C05493=1186.464,-67.586,-41.401,179.419,5.670,149.176
C05494=1186.458,-67.337,-41.411,179.422,5.670,149.175
C05495=1186.453,-67.087,-41.423,179.424,5.671,149.175
C05496=1186.448,-66.837,-41.433,179.426,5.671,149.174
C05497=1186.442,-66.588,-41.445,179.429,5.671,149.173
C05498=1186.438,-66.338,-41.456,179.431,5.672,149.173
C05499=1186.432,-66.088,-41.466,179.433,5.672,149.172
C05500=1186.427,-65.839,-41.477,179.436,5.672,149.171
C05501=1186.422,-65.589,-41.489,179.438,5.673,149.171
C05502=1186.416,-65.339,-41.500,179.440,5.672,149.170
C05503=1186.412,-65.090,-41.511,179.443,5.673,149.169
C05504=1186.406,-64.839,-41.522,179.445,5.674,149.169
C05505=1186.401,-64.590,-41.533,179.447,5.673,149.168
C05506=1186.396,-64.341,-41.544,179.450,5.674,149.168
C05507=1186.391,-64.090,-41.555,179.452,5.675,149.167
C05508=1186.385,-63.841,-41.566,179.454,5.674,149.166
C05509=1186.380,-63.591,-41.578,179.457,5.675,149.166
C05510=1186.376,-63.342,-41.589,179.459,5.675,149.165
C05511=1186.369,-63.092,-41.600,179.461,5.675,149.164
C05512=1186.365,-62.842,-41.611,179.464,5.675,149.164
C05513=1186.360,-62.593,-41.622,179.466,5.676,149.163
C05514=1186.354,-62.342,-41.633,179.468,5.676,149.163
C05515=1186.349,-62.093,-41.644,179.471,5.676,149.162
C05516=1186.344,-61.844,-41.656,179.473,5.677,149.161
C05517=1186.339,-61.594,-41.668,179.475,5.677,149.161
C05518=1186.333,-61.344,-41.678,179.478,5.677,149.160
C05519=1186.328,-61.094,-41.690,179.480,5.678,149.159
C05520=1186.323,-60.845,-41.701,179.482,5.677,149.159
C05521=1186.318,-60.595,-41.712,179.485,5.678,149.158
C05522=1186.312,-60.345,-41.723,179.487,5.678,149.157
C05523=1186.307,-60.095,-41.734,179.489,5.678,149.157
C05524=1186.302,-59.846,-41.746,179.491,5.679,149.156
C05525=1186.297,-59.596,-41.757,179.494,5.679,149.156
C05526=1186.292,-59.347,-41.768,179.497,5.680,149.155
C05527=1186.286,-59.096,-41.780,179.498,5.680,149.154
C05528=1186.281,-58.847,-41.791,179.501,5.680,149.154
C05529=1186.275,-58.598,-41.802,179.504,5.681,149.153
C05530=1186.271,-58.348,-41.814,179.506,5.680,149.152
C05531=1186.266,-58.098,-41.825,179.508,5.681,149.152
C05532=1186.261,-57.848,-41.837,179.511,5.681,149.151
C05533=1186.256,-57.598,-41.847,179.513,5.681,149.150
C05534=1186.250,-57.349,-41.859,179.515,5.682,149.150
C05535=1186.245,-57.099,-41.870,179.518,5.682,149.149
C05536=1186.239,-56.849,-41.882,179.520,5.683,149.148
C05537=1186.235,-56.600,-41.893,179.522,5.683,149.148
C05538=1186.229,-56.351,-41.905,179.525,5.683,149.147
C05539=1186.224,-56.101,-41.916,179.527,5.684,149.147
C05540=1186.219,-55.851,-41.928,179.529,5.683,149.146
C05541=1186.214,-55.601,-41.939,179.531,5.684,149.145
C05542=1186.209,-55.352,-41.951,179.534,5.685,149.145
C05543=1186.203,-55.102,-41.961,179.536,5.684,149.144
C05544=1186.198,-54.852,-41.973,179.538,5.685,149.144
C05545=1186.193,-54.602,-41.985,179.541,5.685,149.143
C05546=1186.188,-54.353,-41.996,179.544,5.686,149.142
C05547=1186.183,-54.103,-42.008,179.546,5.685,149.141
C05548=1186.178,-53.853,-42.019,179.548,5.686,149.141
C05549=1186.172,-53.604,-42.031,179.551,5.687,149.140
C05550=1186.166,-53.354,-42.043,179.553,5.686,149.140
C05551=1186.162,-53.104,-42.054,179.555,5.687,149.139
C05552=1186.156,-52.854,-42.066,179.558,5.688,149.138
C05553=1186.152,-52.605,-42.077,179.560,5.688,149.138
C05554=1186.146,-52.355,-42.089,179.562,5.688,149.137
C05555=1186.141,-52.106,-42.100,179.564,5.688,149.136
C05556=1186.136,-51.856,-42.112,179.567,5.689,149.136
C05557=1186.131,-51.606,-42.123,179.569,5.689,149.135
C05558=1186.125,-51.356,-42.135,179.571,5.689,149.135
C05559=1186.120,-51.106,-42.147,179.574,5.690,149.134
C05560=1186.115,-50.857,-42.158,179.577,5.690,149.133
C05561=1186.110,-50.607,-42.171,179.579,5.690,149.132
C05562=1186.105,-50.359,-42.182,179.581,5.691,149.132
C05563=1186.099,-50.109,-42.193,179.584,5.691,149.131
C05564=1186.094,-49.838,-42.206,179.586,5.692,149.131
C05565=1186.088,-49.568,-42.218,179.589,5.692,149.130
C05566=1186.083,-49.298,-42.231,179.591,5.692,149.129
C05567=1186.077,-49.027,-42.244,179.594,5.692,149.128
C05568=1186.072,-48.777,-42.256,179.596,5.693,149.128
C05569=1186.067,-48.528,-42.267,179.599,5.693,149.127
C05570=1186.061,-48.278,-42.279,179.601,5.693,149.127
C05571=1186.056,-48.029,-42.291,179.603,5.693,149.126
C05572=1186.051,-47.779,-42.302,179.606,5.694,149.125
C05573=1186.046,-47.529,-42.314,179.608,5.695,149.125
C05574=1186.040,-47.280,-42.327,179.610,5.694,149.124
C05575=1186.036,-47.030,-42.338,179.613,5.695,149.123
C05576=1186.030,-46.780,-42.350,179.615,5.696,149.123
C05577=1186.025,-46.530,-42.362,179.618,5.696,149.122
C05578=1186.020,-46.281,-42.373,179.620,5.696,149.121
C05579=1186.015,-46.031,-42.386,179.622,5.696,149.121
C05580=1186.010,-45.781,-42.397,179.625,5.697,149.120
C05581=1186.004,-45.532,-42.408,179.627,5.697,149.120
C05582=1185.999,-45.282,-42.420,179.629,5.697,149.119
C05583=1185.994,-45.033,-42.432,179.632,5.698,149.118
C05584=1185.988,-44.783,-42.445,179.634,5.698,149.118
C05585=1185.984,-44.534,-42.456,179.637,5.699,149.117
C05586=1185.978,-44.284,-42.468,179.639,5.699,149.116
C05587=1185.973,-44.034,-42.480,179.641,5.699,149.116
C05588=1185.968,-43.784,-42.492,179.644,5.700,149.115
C05589=1185.963,-43.535,-42.504,179.647,5.700,149.114
C05590=1185.958,-43.285,-42.516,179.648,5.700,149.114
C05591=1185.952,-43.035,-42.528,179.651,5.700,149.113
C05592=1185.947,-42.786,-42.540,179.653,5.701,149.113
C05593=1185.942,-42.536,-42.551,179.656,5.701,149.112
C05594=1185.937,-42.286,-42.563,179.658,5.701,149.111
C05595=1185.932,-42.037,-42.576,179.660,5.702,149.111
C05596=1185.926,-41.787,-42.588,179.663,5.702,149.110
C05597=1185.922,-41.537,-42.599,179.665,5.703,149.109
C05598=1185.917,-41.288,-42.612,179.667,5.703,149.109
C05599=1185.911,-41.038,-42.623,179.670,5.703,149.108
C05600=1185.906,-40.788,-42.635,179.673,5.704,149.107
C05601=1185.901,-40.539,-42.648,179.675,5.704,149.107
C05602=1185.896,-40.289,-42.659,179.677,5.705,149.106
C05603=1185.891,-40.040,-42.672,179.680,5.704,149.105
C05604=1185.885,-39.790,-42.684,179.682,5.705,149.105
C05605=1185.880,-39.540,-42.696,179.684,5.706,149.104
C05606=1185.875,-39.290,-42.708,179.687,5.706,149.104
C05607=1185.869,-39.041,-42.720,179.689,5.706,149.103
C05608=1185.865,-38.792,-42.732,179.691,5.707,149.102
C05609=1185.860,-38.542,-42.744,179.694,5.707,149.102
C05610=1185.854,-38.292,-42.756,179.697,5.708,149.101
C05611=1185.849,-38.042,-42.768,179.699,5.708,149.100
C05612=1185.844,-37.792,-42.780,179.701,5.708,149.100
C05613=1185.838,-37.543,-42.793,179.704,5.708,149.099
C05614=1185.833,-37.293,-42.805,179.706,5.709,149.098
C05615=1185.828,-37.044,-42.817,179.709,5.709,149.098
C05616=1185.823,-36.794,-42.829,179.710,5.709,149.097
C05617=1185.818,-36.545,-42.841,179.713,5.710,149.097
C05618=1185.813,-36.294,-42.854,179.716,5.710,149.096
C05619=1185.808,-36.045,-42.866,179.718,5.711,149.095
C05620=1185.803,-35.795,-42.878,179.721,5.711,149.095
C05621=1185.798,-35.546,-42.891,179.723,5.711,149.094
C05622=1185.792,-35.296,-42.903,179.725,5.712,149.093
C05623=1185.787,-35.046,-42.915,179.728,5.712,149.093
C05624=1185.782,-34.796,-42.927,179.730,5.713,149.092
C05625=1185.776,-34.547,-42.940,179.733,5.713,149.091
C05626=1185.771,-34.297,-42.952,179.735,5.713,149.091
C05627=1185.766,-34.048,-42.964,179.737,5.714,149.090
C05628=1185.760,-33.798,-42.976,179.740,5.714,149.090
C05629=1185.755,-33.549,-42.989,179.742,5.715,149.089
C05630=1185.751,-33.299,-43.002,179.745,5.715,149.088
C05631=1185.745,-33.049,-43.013,179.747,5.715,149.088
C05632=1185.740,-32.799,-43.026,179.749,5.716,149.087
C05633=1185.735,-32.549,-43.038,179.752,5.716,149.086
C05634=1185.730,-32.300,-43.051,179.754,5.717,149.086
C05635=1185.725,-32.051,-43.063,179.757,5.717,149.085
C05636=1185.719,-31.801,-43.075,179.759,5.717,149.084
C05637=1185.714,-31.552,-43.088,179.762,5.717,149.084
C05638=1185.709,-31.302,-43.101,179.764,5.718,149.083
C05639=1185.704,-31.052,-43.112,179.766,5.719,149.083
C05640=1185.699,-30.802,-43.125,179.769,5.719,149.082
C05641=1185.694,-30.553,-43.138,179.771,5.719,149.081
C05642=1185.688,-30.303,-43.150,179.773,5.720,149.081
C05643=1185.683,-30.054,-43.162,179.776,5.720,149.080
C05644=1185.679,-29.804,-43.175,179.779,5.721,149.079
C05645=1185.673,-29.554,-43.187,179.781,5.721,149.079
C05646=1185.668,-29.304,-43.200,179.783,5.721,149.078
C05647=1185.663,-29.055,-43.212,179.786,5.721,149.077
C05648=1185.658,-28.805,-43.224,179.788,5.722,149.077
C05649=1185.653,-28.556,-43.237,179.790,5.723,149.076
C05650=1185.648,-28.306,-43.250,179.793,5.723,149.076
C05651=1185.643,-28.057,-43.262,179.796,5.724,149.075
C05652=1185.637,-27.807,-43.274,179.798,5.723,149.074
C05653=1185.632,-27.557,-43.287,179.800,5.724,149.074
C05654=1185.627,-27.308,-43.299,179.803,5.725,149.073
C05655=1185.622,-27.058,-43.313,179.805,5.725,149.072
C05656=1185.617,-26.808,-43.326,179.808,5.725,149.072
C05657=1185.611,-26.558,-43.337,179.810,5.726,149.071
C05658=1185.606,-26.309,-43.350,179.812,5.726,149.070
C05659=1185.601,-26.060,-43.363,179.815,5.726,149.070
C05660=1185.597,-25.810,-43.376,179.818,5.727,149.069
C05661=1185.591,-25.560,-43.388,179.820,5.728,149.069
C05662=1185.586,-25.310,-43.400,179.822,5.728,149.068
C05663=1185.581,-25.061,-43.413,179.825,5.729,149.067
C05664=1185.576,-24.811,-43.426,179.827,5.729,149.067
C05665=1185.571,-24.562,-43.439,179.829,5.729,149.066
C05666=1185.565,-24.312,-43.451,179.832,5.730,149.065
C05667=1185.560,-24.063,-43.464,179.835,5.730,149.065
C05668=1185.555,-23.793,-43.478,179.837,5.730,149.064
C05669=1185.550,-23.523,-43.492,179.840,5.731,149.063
C05670=1185.544,-23.253,-43.505,179.843,5.731,149.063
C05671=1185.538,-22.983,-43.519,179.845,5.732,149.062
C05672=1185.533,-22.734,-43.531,179.847,5.733,149.061
C05673=1185.528,-22.484,-43.544,179.850,5.733,149.061
C05674=1185.523,-22.235,-43.557,179.852,5.733,149.060
C05675=1185.517,-21.985,-43.570,179.854,5.734,149.060
C05676=1185.512,-21.736,-43.583,179.857,5.734,149.059
C05677=1185.508,-21.486,-43.596,179.860,5.735,149.058
C05678=1185.503,-21.236,-43.608,179.862,5.735,149.057
C05679=1185.497,-20.987,-43.622,179.865,5.736,149.057
C05680=1185.492,-20.737,-43.635,179.867,5.735,149.056
C05681=1185.487,-20.488,-43.647,179.869,5.736,149.056
C05682=1185.482,-20.238,-43.660,179.872,5.736,149.055
C05683=1185.476,-19.989,-43.673,179.874,5.737,149.054
C05684=1185.471,-19.739,-43.686,179.877,5.738,149.054
C05685=1185.466,-19.489,-43.699,179.879,5.738,149.053
C05686=1185.461,-19.240,-43.712,179.882,5.739,149.053
C05687=1185.456,-18.990,-43.725,179.884,5.739,149.052
C05688=1185.451,-18.740,-43.737,179.886,5.739,149.051
C05689=1185.446,-18.491,-43.750,179.889,5.740,149.051
C05690=1185.440,-18.241,-43.763,179.891,5.740,149.050
C05691=1185.435,-17.991,-43.776,179.894,5.741,149.049
C05692=1185.430,-17.742,-43.789,179.896,5.741,149.049
C05693=1185.425,-17.492,-43.802,179.899,5.742,149.048
C05694=1185.420,-17.242,-43.815,179.901,5.743,149.047
C05695=1185.415,-16.993,-43.827,179.903,5.742,149.047
C05696=1185.409,-16.743,-43.841,179.906,5.743,149.046
C05697=1185.405,-16.494,-43.854,179.909,5.743,149.045
C05698=1185.400,-16.245,-43.867,179.911,5.744,149.045
C05699=1185.394,-15.994,-43.880,179.914,5.744,149.044
C05700=1185.389,-15.745,-43.893,179.916,5.745,149.044
C05701=1185.385,-15.495,-43.906,179.918,5.746,149.043
C05702=1185.379,-15.245,-43.919,179.921,5.746,149.042
C05703=1185.374,-14.996,-43.932,179.924,5.747,149.042
C05704=1185.369,-14.746,-43.946,179.926,5.746,149.041
C05705=1185.364,-14.497,-43.959,179.928,5.747,149.041
C05706=1185.358,-14.248,-43.971,179.931,5.748,149.040
C05707=1185.353,-13.997,-43.985,179.933,5.748,149.039
C05708=1185.348,-13.748,-43.997,179.936,5.749,149.038
C05709=1185.344,-13.498,-44.010,179.938,5.749,149.038
C05710=1185.338,-13.249,-44.024,179.941,5.750,149.037
C05711=1185.333,-13.000,-44.037,179.943,5.750,149.037
C05712=1185.328,-12.749,-44.051,179.946,5.751,149.036
C05713=1185.322,-12.500,-44.063,179.948,5.751,149.035
C05714=1185.317,-12.250,-44.077,179.950,5.751,149.035
C05715=1185.312,-12.001,-44.090,179.953,5.752,149.034
C05716=1185.308,-11.751,-44.103,179.955,5.753,149.034
C05717=1185.302,-11.501,-44.116,179.958,5.753,149.033
C05718=1185.297,-11.253,-44.129,179.960,5.754,149.032
C05719=1185.292,-11.002,-44.143,179.963,5.754,149.032
C05720=1185.287,-10.753,-44.156,179.965,5.755,149.031
C05721=1185.282,-10.503,-44.170,179.968,5.755,149.030
C05722=1185.277,-10.254,-44.183,179.971,5.756,149.030
C05723=1185.271,-10.004,-44.196,179.973,5.755,149.029
C05724=1185.266,-9.754,-44.209,179.975,5.756,149.029
C05725=1185.261,-9.505,-44.223,179.977,5.757,149.028
C05726=1185.256,-9.255,-44.236,179.980,5.757,149.027
C05727=1185.251,-9.005,-44.249,179.983,5.758,149.026
C05728=1185.246,-8.756,-44.262,179.985,5.759,149.026
C05729=1185.241,-8.506,-44.276,179.988,5.759,149.025
C05730=1185.236,-8.257,-44.289,179.990,5.759,149.025
C05731=1185.231,-8.007,-44.303,179.992,5.760,149.024
C05732=1185.226,-7.758,-44.315,179.995,5.761,149.023
C05733=1185.221,-7.508,-44.330,179.998,5.761,149.023
C05734=1185.216,-7.259,-44.342,180.000,5.761,149.022
C05735=1185.211,-7.009,-44.357,-179.998,5.762,149.022
C05736=1185.206,-6.760,-44.369,-179.995,5.762,149.021
C05737=1185.200,-6.509,-44.383,-179.993,5.763,149.020
C05738=1185.195,-6.260,-44.397,-179.990,5.763,149.020
C05739=1185.190,-6.010,-44.410,-179.988,5.764,149.019
C05740=1185.185,-5.761,-44.424,-179.985,5.765,149.018
C05741=1185.180,-5.511,-44.437,-179.983,5.765,149.018
C05742=1185.175,-5.262,-44.450,-179.980,5.766,149.017
C05743=1185.169,-5.012,-44.464,-179.978,5.766,149.017
C05744=1185.164,-4.763,-44.477,-179.975,5.767,149.016
C05745=1185.159,-4.513,-44.491,-179.972,5.767,149.015
C05746=1185.154,-4.264,-44.504,-179.970,5.768,149.015
C05747=1185.149,-4.014,-44.518,-179.968,5.769,149.014
C05748=1185.144,-3.765,-44.532,-179.965,5.769,149.013
C05749=1185.139,-3.515,-44.545,-179.963,5.769,149.013
C05750=1185.134,-3.265,-44.559,-179.961,5.770,149.012
C05751=1185.128,-3.015,-44.572,-179.958,5.770,149.011
C05752=1185.124,-2.766,-44.586,-179.955,5.770,149.011
C05753=1185.118,-2.516,-44.599,-179.953,5.771,149.010
C05754=1185.113,-2.267,-44.613,-179.951,5.772,149.010
C05755=1185.108,-2.017,-44.626,-179.948,5.772,149.009
C05756=1185.103,-1.768,-44.640,-179.945,5.773,149.008
C05757=1185.098,-1.518,-44.654,-179.943,5.774,149.008
C05758=1185.093,-1.269,-44.667,-179.940,5.774,149.007
C05759=1185.088,-1.019,-44.681,-179.938,5.775,149.006
C05760=1185.082,-0.769,-44.695,-179.935,5.775,149.006
C05761=1185.078,-0.520,-44.708,-179.933,5.776,149.005
C05762=1185.073,-0.270,-44.722,-179.930,5.776,149.005
C05763=1185.067,-0.021,-44.736,-179.928,5.777,149.004
C05764=1185.062,0.229,-44.750,-179.925,5.778,149.003
C05765=1185.057,0.478,-44.763,-179.923,5.778,149.003
C05766=1185.052,0.728,-44.777,-179.920,5.779,149.002
C05767=1185.047,0.978,-44.791,-179.918,5.779,149.001
C05768=1185.042,1.227,-44.804,-179.915,5.780,149.001
C05769=1185.037,1.477,-44.818,-179.913,5.780,149.000
C05770=1185.032,1.727,-44.832,-179.911,5.780,149.000
C05771=1185.027,1.976,-44.846,-179.908,5.781,148.999
C05772=1185.021,2.245,-44.861,-179.905,5.782,148.998
C05773=1185.016,2.514,-44.876,-179.903,5.783,148.998
C05774=1185.011,2.784,-44.891,-179.900,5.783,148.997
C05775=1185.005,3.052,-44.905,-179.897,5.784,148.996
C05776=1185.000,3.302,-44.919,-179.895,5.784,148.996
C05777=1184.995,3.552,-44.933,-179.892,5.785,148.995
C05778=1184.989,3.801,-44.947,-179.890,5.785,148.994
C05779=1184.984,4.051,-44.961,-179.887,5.786,148.994
C05780=1184.980,4.300,-44.975,-179.884,5.786,148.993
C05781=1184.975,4.549,-44.989,-179.882,5.787,148.992
C05782=1184.969,4.800,-45.002,-179.880,5.788,148.992
C05783=1184.964,5.049,-45.017,-179.877,5.788,148.991
C05784=1184.959,5.298,-45.031,-179.874,5.789,148.991
C05785=1184.954,5.548,-45.045,-179.872,5.790,148.990
C05786=1184.950,5.798,-45.058,-179.870,5.790,148.989
C05787=1184.944,6.047,-45.072,-179.867,5.791,148.989
C05788=1184.939,6.297,-45.086,-179.864,5.791,148.988
C05789=1184.934,6.547,-45.100,-179.862,5.792,148.988
C05790=1184.929,6.796,-45.115,-179.859,5.792,148.987
C05791=1184.923,7.045,-45.128,-179.857,5.793,148.986
C05792=1184.918,7.295,-45.143,-179.855,5.794,148.986
C05793=1184.913,7.545,-45.157,-179.852,5.794,148.985
C05794=1184.909,7.794,-45.171,-179.849,5.795,148.984
C05795=1184.904,8.043,-45.185,-179.847,5.795,148.984
C05796=1184.898,8.294,-45.198,-179.844,5.796,148.983
C05797=1184.893,8.543,-45.212,-179.842,5.796,148.983
C05798=1184.888,8.792,-45.226,-179.839,5.797,148.982
C05799=1184.883,9.042,-45.241,-179.837,5.798,148.981
C05800=1184.878,9.292,-45.255,-179.834,5.798,148.981
C05801=1184.873,9.541,-45.269,-179.832,5.799,148.980
C05802=1184.868,9.791,-45.283,-179.829,5.799,148.979
C05803=1184.862,10.040,-45.297,-179.827,5.800,148.979
C05804=1184.858,10.290,-45.312,-179.824,5.801,148.978
C05805=1184.853,10.540,-45.326,-179.822,5.801,148.978
C05806=1184.848,10.789,-45.340,-179.819,5.802,148.977
C05807=1184.842,11.038,-45.354,-179.817,5.802,148.976
C05808=1184.837,11.288,-45.368,-179.814,5.803,148.976
C05809=1184.832,11.538,-45.383,-179.812,5.804,148.975
C05810=1184.827,11.787,-45.397,-179.809,5.804,148.975
C05811=1184.822,12.037,-45.411,-179.807,5.805,148.974
C05812=1184.817,12.286,-45.425,-179.804,5.805,148.973
C05813=1184.812,12.536,-45.439,-179.802,5.806,148.973
C05814=1184.807,12.786,-45.454,-179.799,5.807,148.972
C05815=1184.802,13.035,-45.468,-179.797,5.807,148.971
C05816=1184.797,13.285,-45.482,-179.794,5.808,148.971
C05817=1184.791,13.534,-45.496,-179.792,5.808,148.970
C05818=1184.787,13.783,-45.511,-179.789,5.809,148.970
C05819=1184.782,14.033,-45.525,-179.786,5.809,148.969
C05820=1184.777,14.282,-45.540,-179.784,5.810,148.968
C05821=1184.772,14.532,-45.554,-179.782,5.811,148.968
C05822=1184.767,14.782,-45.568,-179.779,5.811,148.967
C05823=1184.761,15.031,-45.582,-179.777,5.812,148.967
C05824=1184.756,15.281,-45.596,-179.774,5.812,148.966
C05825=1184.751,15.530,-45.611,-179.772,5.813,148.965
C05826=1184.747,15.779,-45.626,-179.769,5.814,148.965
C05827=1184.742,16.029,-45.640,-179.767,5.814,148.964
C05828=1184.737,16.279,-45.654,-179.764,5.815,148.963
C05829=1184.731,16.528,-45.669,-179.761,5.815,148.963
C05830=1184.726,16.778,-45.683,-179.759,5.816,148.962
C05831=1184.721,17.027,-45.698,-179.757,5.817,148.962
C05832=1184.716,17.277,-45.712,-179.754,5.817,148.961
C05833=1184.711,17.526,-45.727,-179.751,5.819,148.960
C05834=1184.706,17.776,-45.741,-179.749,5.819,148.960
C05835=1184.701,18.026,-45.755,-179.746,5.820,148.959
C05836=1184.696,18.275,-45.770,-179.744,5.821,148.959
C05837=1184.691,18.525,-45.785,-179.741,5.821,148.958
C05838=1184.685,18.774,-45.799,-179.738,5.822,148.957
C05839=1184.681,19.023,-45.814,-179.736,5.822,148.957
C05840=1184.676,19.273,-45.828,-179.734,5.823,148.956
C05841=1184.671,19.522,-45.842,-179.731,5.823,148.955
C05842=1184.666,19.772,-45.857,-179.728,5.824,148.955
C05843=1184.660,20.022,-45.872,-179.726,5.825,148.954
C05844=1184.655,20.271,-45.887,-179.724,5.825,148.954
C05845=1184.650,20.521,-45.901,-179.721,5.826,148.953
C05846=1184.646,20.770,-45.916,-179.719,5.827,148.953
C05847=1184.641,21.020,-45.930,-179.716,5.827,148.952
C05848=1184.635,21.270,-45.945,-179.713,5.828,148.951
C05849=1184.630,21.519,-45.960,-179.711,5.829,148.951
C05850=1184.626,21.769,-45.974,-179.708,5.830,148.950
C05851=1184.621,22.018,-45.989,-179.705,5.830,148.949
C05852=1184.615,22.268,-46.004,-179.703,5.831,148.949
C05853=1184.610,22.517,-46.018,-179.701,5.832,148.948
C05854=1184.605,22.766,-46.033,-179.698,5.832,148.948
C05855=1184.600,23.015,-46.047,-179.695,5.833,148.947
C05856=1184.594,23.266,-46.062,-179.693,5.834,148.946
C05857=1184.590,23.515,-46.077,-179.690,5.834,148.946
C05858=1184.585,23.764,-46.091,-179.688,5.834,148.945
C05859=1184.580,24.013,-46.106,-179.686,5.835,148.945
C05860=1184.574,24.263,-46.121,-179.683,5.836,148.944
C05861=1184.570,24.513,-46.136,-179.680,5.836,148.943
C05862=1184.565,24.762,-46.151,-179.678,5.838,148.943
C05863=1184.559,25.012,-46.166,-179.675,5.839,148.942
C05864=1184.554,25.261,-46.180,-179.672,5.839,148.941
C05865=1184.550,25.510,-46.195,-179.670,5.840,148.941
C05866=1184.545,25.760,-46.210,-179.668,5.840,148.940
C05867=1184.539,26.010,-46.225,-179.665,5.841,148.940
C05868=1184.534,26.259,-46.240,-179.663,5.842,148.939
C05869=1184.530,26.508,-46.255,-179.660,5.842,148.938
C05870=1184.524,26.758,-46.269,-179.657,5.843,148.938
C05871=1184.519,27.007,-46.284,-179.655,5.844,148.937
C05872=1184.514,27.257,-46.299,-179.653,5.844,148.937
C05873=1184.510,27.507,-46.315,-179.649,5.845,148.936
C05874=1184.505,27.757,-46.329,-179.647,5.846,148.935
C05875=1184.499,28.006,-46.345,-179.645,5.847,148.935
C05876=1184.494,28.275,-46.360,-179.642,5.847,148.934
C05877=1184.488,28.544,-46.377,-179.639,5.848,148.933
C05878=1184.484,28.812,-46.393,-179.636,5.849,148.933
C05879=1184.478,29.082,-46.409,-179.633,5.850,148.932
C05880=1184.473,29.331,-46.424,-179.631,5.850,148.932
C05881=1184.468,29.580,-46.439,-179.629,5.851,148.931
C05882=1184.463,29.830,-46.454,-179.626,5.851,148.930
C05883=1184.458,30.079,-46.468,-179.624,5.852,148.930
C05884=1184.452,30.329,-46.484,-179.621,5.853,148.929
C05885=1184.448,30.578,-46.499,-179.618,5.854,148.929
C05886=1184.442,30.828,-46.514,-179.616,5.855,148.928
C05887=1184.437,31.077,-46.529,-179.613,5.855,148.927
C05888=1184.433,31.326,-46.544,-179.610,5.856,148.927
C05889=1184.427,31.576,-46.559,-179.608,5.857,148.926
C05890=1184.423,31.826,-46.574,-179.606,5.857,148.926
C05891=1184.418,32.075,-46.590,-179.603,5.858,148.925
C05892=1184.413,32.324,-46.605,-179.601,5.859,148.924
C05893=1184.407,32.575,-46.620,-179.598,5.860,148.924
C05894=1184.403,32.824,-46.635,-179.595,5.861,148.923
C05895=1184.397,33.073,-46.650,-179.593,5.861,148.923
C05896=1184.393,33.322,-46.665,-179.590,5.862,148.922
C05897=1184.387,33.572,-46.680,-179.588,5.862,148.921
C05898=1184.383,33.822,-46.695,-179.585,5.863,148.921
C05899=1184.377,34.071,-46.711,-179.583,5.864,148.920
C05900=1184.373,34.320,-46.726,-179.580,5.864,148.920
C05901=1184.367,34.570,-46.742,-179.577,5.866,148.919
C05902=1184.362,34.820,-46.756,-179.575,5.866,148.918
C05903=1184.357,35.069,-46.771,-179.572,5.867,148.918
C05904=1184.352,35.318,-46.787,-179.570,5.868,148.917
C05905=1184.348,35.568,-46.802,-179.567,5.868,148.917
C05906=1184.342,35.818,-46.818,-179.565,5.869,148.916
C05907=1184.338,36.067,-46.833,-179.562,5.870,148.915
C05908=1184.332,36.317,-46.848,-179.559,5.871,148.915
C05909=1184.327,36.566,-46.863,-179.557,5.872,148.914
C05910=1184.322,36.816,-46.879,-179.554,5.872,148.914
C05911=1184.317,37.065,-46.894,-179.552,5.873,148.913
C05912=1184.312,37.314,-46.909,-179.549,5.873,148.912
C05913=1184.307,37.564,-46.925,-179.547,5.874,148.912
C05914=1184.302,37.813,-46.940,-179.544,5.876,148.911
C05915=1184.298,38.063,-46.956,-179.541,5.876,148.911
C05916=1184.292,38.312,-46.971,-179.539,5.877,148.910
C05917=1184.288,38.561,-46.986,-179.536,5.877,148.909
C05918=1184.282,38.811,-47.002,-179.534,5.878,148.909
C05919=1184.277,39.060,-47.018,-179.532,5.879,148.908
C05920=1184.273,39.310,-47.033,-179.528,5.880,148.908
C05921=1184.267,39.559,-47.049,-179.526,5.881,148.907
C05922=1184.262,39.809,-47.064,-179.524,5.882,148.907
C05923=1184.257,40.058,-47.079,-179.521,5.882,148.906
C05924=1184.253,40.308,-47.095,-179.519,5.883,148.905
C05925=1184.247,40.557,-47.111,-179.516,5.883,148.905
C05926=1184.242,40.807,-47.126,-179.513,5.885,148.904
C05927=1184.237,41.056,-47.141,-179.511,5.886,148.904
C05928=1184.232,41.306,-47.157,-179.508,5.886,148.903
C05929=1184.227,41.555,-47.173,-179.505,5.887,148.902
C05930=1184.222,41.804,-47.188,-179.503,5.888,148.902
C05931=1184.217,42.054,-47.203,-179.501,5.888,148.901
C05932=1184.212,42.304,-47.219,-179.497,5.889,148.900
C05933=1184.207,42.553,-47.235,-179.495,5.890,148.900
C05934=1184.202,42.802,-47.250,-179.493,5.891,148.899
C05935=1184.197,43.053,-47.266,-179.490,5.892,148.899
C05936=1184.192,43.302,-47.281,-179.488,5.892,148.898
C05937=1184.187,43.551,-47.297,-179.485,5.893,148.898
C05938=1184.182,43.800,-47.313,-179.482,5.894,148.897
C05939=1184.177,44.050,-47.329,-179.480,5.895,148.896
C05940=1184.172,44.299,-47.344,-179.477,5.895,148.896
C05941=1184.167,44.549,-47.360,-179.475,5.896,148.895
C05942=1184.163,44.799,-47.375,-179.472,5.898,148.895
C05943=1184.157,45.048,-47.391,-179.469,5.898,148.894
C05944=1184.152,45.297,-47.407,-179.467,5.899,148.894
C05945=1184.147,45.547,-47.423,-179.464,5.899,148.893
C05946=1184.142,45.796,-47.439,-179.462,5.900,148.892
C05947=1184.137,46.046,-47.454,-179.459,5.902,148.892
C05948=1184.133,46.295,-47.470,-179.456,5.902,148.891
C05949=1184.127,46.544,-47.486,-179.454,5.903,148.891
C05950=1184.122,46.794,-47.502,-179.452,5.904,148.890
C05951=1184.117,47.044,-47.517,-179.449,5.904,148.889
C05952=1184.112,47.293,-47.533,-179.446,5.906,148.889
C05953=1184.107,47.542,-47.549,-179.444,5.906,148.888
C05954=1184.103,47.792,-47.565,-179.441,5.907,148.888
C05955=1184.097,48.041,-47.580,-179.439,5.908,148.887
C05956=1184.093,48.291,-47.597,-179.436,5.909,148.886
C05957=1184.088,48.540,-47.613,-179.433,5.910,148.886
C05958=1184.082,48.789,-47.628,-179.431,5.910,148.885
C05959=1184.077,49.040,-47.644,-179.428,5.911,148.885
C05960=1184.072,49.288,-47.660,-179.426,5.912,148.884
C05961=1184.067,49.538,-47.676,-179.423,5.913,148.884
C05962=1184.062,49.787,-47.693,-179.421,5.914,148.883
C05963=1184.058,50.036,-47.708,-179.418,5.915,148.882
C05964=1184.053,50.286,-47.724,-179.415,5.915,148.882
C05965=1184.048,50.535,-47.740,-179.413,5.917,148.881
C05966=1184.043,50.785,-47.756,-179.410,5.917,148.881
C05967=1184.038,51.035,-47.771,-179.408,5.918,148.880
C05968=1184.033,51.283,-47.788,-179.405,5.919,148.880
C05969=1184.028,51.534,-47.804,-179.402,5.920,148.879
C05970=1184.023,51.782,-47.820,-179.400,5.921,148.878
C05971=1184.018,52.032,-47.836,-179.397,5.921,148.878
C05972=1184.013,52.281,-47.852,-179.395,5.922,148.877
C05973=1184.008,52.531,-47.868,-179.392,5.923,148.877
C05974=1184.003,52.781,-47.884,-179.389,5.924,148.876
C05975=1183.998,53.030,-47.900,-179.387,5.925,148.876
C05976=1183.993,53.280,-47.916,-179.384,5.925,148.875
C05977=1183.988,53.529,-47.933,-179.382,5.926,148.874
C05978=1183.983,53.779,-47.948,-179.379,5.928,148.874
C05979=1183.978,54.027,-47.965,-179.376,5.928,148.873
C05980=1183.973,54.296,-47.982,-179.374,5.929,148.872
C05981=1183.967,54.565,-47.999,-179.371,5.930,148.872
C05982=1183.962,54.833,-48.017,-179.368,5.931,148.871
C05983=1183.957,55.102,-48.034,-179.365,5.932,148.871
C05984=1183.952,55.351,-48.050,-179.362,5.933,148.870
C05985=1183.947,55.601,-48.067,-179.360,5.934,148.870
C05986=1183.941,55.850,-48.083,-179.358,5.934,148.869
C05987=1183.937,56.100,-48.099,-179.355,5.936,148.868
C05988=1183.932,56.349,-48.116,-179.352,5.936,148.868
C05989=1183.927,56.599,-48.132,-179.350,5.937,148.867
C05990=1183.922,56.848,-48.148,-179.347,5.939,148.867
C05991=1183.917,57.097,-48.164,-179.344,5.939,148.866
C05992=1183.912,57.347,-48.180,-179.342,5.940,148.866
C05993=1183.907,57.596,-48.197,-179.339,5.941,148.865
C05994=1183.902,57.845,-48.213,-179.337,5.942,148.865
C05995=1183.897,58.095,-48.230,-179.334,5.943,148.864
C05996=1183.892,58.344,-48.246,-179.331,5.943,148.863
C05997=1183.887,58.594,-48.263,-179.329,5.944,148.863
C05998=1183.882,58.843,-48.278,-179.326,5.946,148.862
C05999=1183.877,59.092,-48.295,-179.324,5.946,148.862
C06000=1183.873,59.342,-48.311,-179.321,5.947,148.861
C06001=1183.868,59.591,-48.327,-179.318,5.948,148.860
C06002=1183.862,59.841,-48.344,-179.316,5.949,148.860
C06003=1183.857,60.090,-48.361,-179.313,5.950,148.859
C06004=1183.852,60.340,-48.377,-179.311,5.951,148.859
C06005=1183.847,60.589,-48.393,-179.308,5.952,148.858
C06006=1183.843,60.838,-48.410,-179.306,5.953,148.858
C06007=1183.838,61.088,-48.427,-179.303,5.953,148.857
C06008=1183.832,61.338,-48.442,-179.300,5.955,148.856
C06009=1183.828,61.587,-48.459,-179.298,5.956,148.856
C06010=1183.823,61.836,-48.475,-179.295,5.956,148.855
C06011=1183.818,62.085,-48.492,-179.292,5.958,148.855
C06012=1183.813,62.335,-48.509,-179.290,5.958,148.854
C06013=1183.808,62.584,-48.525,-179.288,5.959,148.854
C06014=1183.803,62.834,-48.542,-179.285,5.960,148.853
C06015=1183.798,63.083,-48.558,-179.282,5.961,148.852
C06016=1183.793,63.333,-48.575,-179.280,5.962,148.852
C06017=1183.788,63.582,-48.592,-179.277,5.962,148.851
C06018=1183.783,63.831,-48.608,-179.274,5.964,148.851
C06019=1183.778,64.081,-48.625,-179.272,5.965,148.850
C06020=1183.773,64.331,-48.641,-179.270,5.966,148.850
C06021=1183.768,64.579,-48.658,-179.266,5.967,148.849
C06022=1183.764,64.829,-48.674,-179.264,5.967,148.848
C06023=1183.758,65.079,-48.692,-179.262,5.968,148.848
C06024=1183.753,65.328,-48.708,-179.258,5.970,148.847
C06025=1183.749,65.577,-48.725,-179.256,5.971,148.847
C06026=1183.744,65.827,-48.742,-179.254,5.971,148.846
C06027=1183.739,66.076,-48.758,-179.251,5.973,148.846
C06028=1183.734,66.325,-48.775,-179.248,5.973,148.845
C06029=1183.729,66.575,-48.792,-179.246,5.974,148.844
C06030=1183.724,66.824,-48.808,-179.243,5.976,148.844
C06031=1183.719,67.073,-48.825,-179.240,5.976,148.843
C06032=1183.714,67.323,-48.842,-179.238,5.977,148.843
C06033=1183.709,67.572,-48.859,-179.235,5.978,148.842
C06034=1183.705,67.821,-48.875,-179.233,5.979,148.842
C06035=1183.699,68.071,-48.893,-179.230,5.980,148.841
C06036=1183.695,68.320,-48.909,-179.227,5.981,148.841
C06037=1183.689,68.570,-48.926,-179.225,5.982,148.840
C06038=1183.685,68.819,-48.943,-179.222,5.983,148.839
C06039=1183.680,69.069,-48.959,-179.219,5.984,148.839
C06040=1183.674,69.318,-48.976,-179.217,5.985,148.838
C06041=1183.670,69.567,-48.993,-179.215,5.986,148.838
C06042=1183.665,69.817,-49.010,-179.211,5.987,148.837
C06043=1183.660,70.066,-49.027,-179.209,5.988,148.837
C06044=1183.655,70.315,-49.043,-179.207,5.988,148.836
C06045=1183.650,70.565,-49.061,-179.204,5.990,148.836
C06046=1183.646,70.814,-49.078,-179.201,5.991,148.835
C06047=1183.640,71.064,-49.095,-179.199,5.992,148.835
C06048=1183.635,71.312,-49.111,-179.196,5.993,148.834
C06049=1183.630,71.562,-49.129,-179.194,5.994,148.834
C06050=1183.626,71.812,-49.145,-179.191,5.994,148.833
C06051=1183.620,72.061,-49.163,-179.188,5.996,148.832
C06052=1183.616,72.311,-49.179,-179.186,5.997,148.832
C06053=1183.610,72.559,-49.197,-179.183,5.998,148.831
C06054=1183.606,72.809,-49.214,-179.180,5.999,148.831
C06055=1183.601,73.059,-49.231,-179.178,5.999,148.830
C06056=1183.596,73.308,-49.248,-179.175,6.001,148.830
C06057=1183.591,73.557,-49.265,-179.172,6.002,148.829
C06058=1183.586,73.806,-49.282,-179.170,6.003,148.829
C06059=1183.581,74.056,-49.299,-179.167,6.004,148.828
C06060=1183.577,74.305,-49.316,-179.165,6.005,148.828
C06061=1183.572,74.555,-49.334,-179.162,6.005,148.827
C06062=1183.566,74.804,-49.351,-179.160,6.007,148.826
C06063=1183.561,75.053,-49.367,-179.157,6.008,148.826
C06064=1183.556,75.303,-49.385,-179.154,6.009,148.825
C06065=1183.552,75.552,-49.402,-179.152,6.010,148.825
C06066=1183.547,75.802,-49.419,-179.149,6.011,148.824
C06067=1183.542,76.051,-49.436,-179.146,6.012,148.824
C06068=1183.537,76.300,-49.454,-179.144,6.013,148.823
C06069=1183.532,76.549,-49.471,-179.141,6.014,148.823
C06070=1183.527,76.799,-49.487,-179.138,6.015,148.822
C06071=1183.522,77.048,-49.505,-179.136,6.016,148.821
C06072=1183.518,77.298,-49.522,-179.133,6.017,148.821
C06073=1183.512,77.547,-49.539,-179.131,6.018,148.820
C06074=1183.508,77.797,-49.557,-179.128,6.019,148.820
C06075=1183.503,78.046,-49.574,-179.125,6.020,148.819
C06076=1183.498,78.294,-49.592,-179.123,6.021,148.819
C06077=1183.492,78.544,-49.609,-179.120,6.022,148.818
C06078=1183.488,78.794,-49.626,-179.117,6.023,148.818
C06079=1183.483,79.043,-49.644,-179.115,6.025,148.817
C06080=1183.478,79.293,-49.661,-179.112,6.025,148.816
C06081=1183.474,79.542,-49.678,-179.110,6.026,148.816
C06082=1183.468,79.791,-49.695,-179.107,6.028,148.815
C06083=1183.463,80.041,-49.713,-179.105,6.028,148.815
C06084=1183.457,80.309,-49.732,-179.101,6.030,148.814
C06085=1183.453,80.577,-49.750,-179.099,6.030,148.814
C06086=1183.448,80.846,-49.769,-179.096,6.032,148.813
C06087=1183.442,81.114,-49.788,-179.093,6.033,148.813
C06088=1183.437,81.364,-49.806,-179.091,6.034,148.812
C06089=1183.433,81.613,-49.823,-179.088,6.035,148.811
C06090=1183.427,81.862,-49.840,-179.085,6.037,148.811
C06091=1183.422,82.111,-49.857,-179.083,6.037,148.810
C06092=1183.417,82.361,-49.875,-179.080,6.039,148.810
C06093=1183.413,82.610,-49.892,-179.077,6.039,148.809
C06094=1183.408,82.859,-49.910,-179.075,6.041,148.809
C06095=1183.403,83.108,-49.928,-179.072,6.042,148.808
C06096=1183.398,83.358,-49.945,-179.070,6.042,148.808
C06097=1183.393,83.607,-49.963,-179.067,6.044,148.807
C06098=1183.388,83.857,-49.980,-179.065,6.045,148.807
C06099=1183.383,84.106,-49.998,-179.061,6.046,148.806
C06100=1183.379,84.355,-50.016,-179.059,6.047,148.806
C06101=1183.373,84.605,-50.033,-179.056,6.048,148.805
C06102=1183.368,84.854,-50.051,-179.054,6.049,148.805
C06103=1183.364,85.103,-50.069,-179.051,6.050,148.804
C06104=1183.359,85.353,-50.086,-179.049,6.052,148.804
C06105=1183.354,85.602,-50.104,-179.046,6.052,148.803
C06106=1183.349,85.851,-50.122,-179.043,6.054,148.802
C06107=1183.344,86.101,-50.139,-179.041,6.054,148.802
C06108=1183.339,86.350,-50.157,-179.038,6.056,148.801
C06109=1183.335,86.599,-50.174,-179.035,6.057,148.801
C06110=1183.330,86.848,-50.192,-179.032,6.058,148.800
C06111=1183.325,87.098,-50.210,-179.030,6.059,148.800
C06112=1183.320,87.347,-50.228,-179.028,6.060,148.799
C06113=1183.315,87.596,-50.246,-179.025,6.061,148.799
C06114=1183.310,87.845,-50.264,-179.022,6.062,148.798
C06115=1183.305,88.095,-50.281,-179.020,6.064,148.798
C06116=1183.300,88.344,-50.299,-179.017,6.064,148.797
C06117=1183.296,88.594,-50.317,-179.014,6.066,148.797
C06118=1183.291,88.844,-50.335,-179.012,6.067,148.796
C06119=1183.286,89.093,-50.353,-179.009,6.068,148.796
C06120=1183.281,89.342,-50.370,-179.006,6.069,148.795
C06121=1183.276,89.591,-50.388,-179.004,6.071,148.795
C06122=1183.271,89.841,-50.406,-179.001,6.071,148.794
C06123=1183.267,90.090,-50.424,-178.998,6.073,148.794
C06124=1183.262,90.339,-50.442,-178.996,6.073,148.793
C06125=1183.257,90.588,-50.460,-178.993,6.075,148.792
C06126=1183.251,90.838,-50.477,-178.991,6.076,148.792
C06127=1183.247,91.087,-50.495,-178.988,6.077,148.791
C06128=1183.242,91.336,-50.513,-178.986,6.078,148.791
C06129=1183.237,91.586,-50.531,-178.983,6.079,148.790
C06130=1183.232,91.835,-50.549,-178.980,6.081,148.790
C06131=1183.228,92.084,-50.567,-178.978,6.081,148.789
C06132=1183.223,92.334,-50.585,-178.975,6.083,148.789
C06133=1183.218,92.583,-50.603,-178.972,6.083,148.788
C06134=1183.213,92.832,-50.621,-178.969,6.085,148.788
C06135=1183.208,93.081,-50.639,-178.967,6.086,148.787
C06136=1183.203,93.330,-50.657,-178.964,6.087,148.787
C06137=1183.198,93.580,-50.676,-178.962,6.088,148.786
C06138=1183.193,93.830,-50.694,-178.959,6.090,148.786
C06139=1183.188,94.079,-50.712,-178.957,6.091,148.785
C06140=1183.183,94.328,-50.730,-178.953,6.092,148.785
C06141=1183.178,94.577,-50.748,-178.951,6.093,148.784
C06142=1183.173,94.826,-50.766,-178.948,6.094,148.784
C06143=1183.169,95.076,-50.784,-178.946,6.095,148.783
C06144=1183.164,95.325,-50.802,-178.943,6.097,148.783
C06145=1183.159,95.575,-50.820,-178.941,6.097,148.782
C06146=1183.154,95.824,-50.838,-178.938,6.099,148.782
C06147=1183.149,96.073,-50.856,-178.935,6.100,148.781
C06148=1183.144,96.322,-50.875,-178.933,6.101,148.781
C06149=1183.140,96.572,-50.894,-178.930,6.102,148.780
C06150=1183.135,96.821,-50.912,-178.927,6.104,148.779
C06151=1183.130,97.070,-50.930,-178.925,6.105,148.779
C06152=1183.125,97.319,-50.948,-178.922,6.106,148.778
C06153=1183.120,97.568,-50.966,-178.919,6.108,148.778
C06154=1183.115,97.819,-50.985,-178.917,6.108,148.777
C06155=1183.110,98.068,-51.003,-178.914,6.110,148.777
C06156=1183.106,98.316,-51.021,-178.912,6.111,148.777
C06157=1183.101,98.565,-51.039,-178.909,6.112,148.776
C06158=1183.096,98.815,-51.058,-178.906,6.113,148.775
C06159=1183.091,99.065,-51.076,-178.903,6.115,148.775
C06160=1183.086,99.314,-51.094,-178.901,6.115,148.774
C06161=1183.081,99.563,-51.113,-178.898,6.117,148.774
C06162=1183.077,99.812,-51.131,-178.896,6.118,148.773
C06163=1183.072,100.062,-51.149,-178.893,6.119,148.773
C06164=1183.066,100.311,-51.168,-178.890,6.120,148.772
C06165=1183.062,100.560,-51.187,-178.888,6.122,148.772
C06166=1183.057,100.810,-51.205,-178.885,6.122,148.771
C06167=1183.052,101.059,-51.223,-178.882,6.124,148.771
C06168=1183.047,101.308,-51.242,-178.880,6.126,148.770
C06169=1183.043,101.557,-51.261,-178.877,6.126,148.770
C06170=1183.038,101.807,-51.279,-178.874,6.128,148.769
C06171=1183.033,102.056,-51.297,-178.872,6.129,148.769
C06172=1183.028,102.305,-51.316,-178.869,6.130,148.768
C06173=1183.023,102.555,-51.334,-178.867,6.131,148.768
C06174=1183.018,102.804,-51.352,-178.864,6.133,148.767
C06175=1183.013,103.053,-51.371,-178.862,6.134,148.767
C06176=1183.009,103.302,-51.390,-178.858,6.135,148.766
C06177=1183.004,103.551,-51.408,-178.856,6.137,148.766
C06178=1182.998,103.801,-51.427,-178.854,6.138,148.765
C06179=1182.994,104.050,-51.445,-178.850,6.139,148.765
C06180=1182.990,104.299,-51.464,-178.848,6.140,148.764
C06181=1182.984,104.548,-51.483,-178.846,6.142,148.764
C06182=1182.980,104.798,-51.502,-178.843,6.142,148.763
C06183=1182.975,105.047,-51.520,-178.840,6.144,148.763
C06184=1182.969,105.296,-51.538,-178.838,6.144,148.762
C06185=1182.965,105.546,-51.557,-178.835,6.146,148.762
C06186=1182.960,105.795,-51.576,-178.832,6.148,148.761
C06187=1182.955,106.044,-51.595,-178.830,6.148,148.761
C06188=1182.950,106.313,-51.615,-178.827,6.150,148.760
C06189=1182.945,106.581,-51.635,-178.824,6.152,148.760
C06190=1182.939,106.849,-51.655,-178.821,6.153,148.759
C06191=1182.935,107.117,-51.676,-178.818,6.154,148.759
C06192=1182.929,107.367,-51.694,-178.816,6.156,148.758
C06193=1182.925,107.616,-51.713,-178.813,6.156,148.758
C06194=1182.920,107.866,-51.732,-178.810,6.158,148.757
C06195=1182.915,108.114,-51.751,-178.808,6.160,148.757
C06196=1182.910,108.364,-51.769,-178.805,6.160,148.756
C06197=1182.906,108.613,-51.788,-178.802,6.162,148.756
C06198=1182.901,108.862,-51.806,-178.800,6.163,148.755
C06199=1182.896,109.112,-51.826,-178.797,6.164,148.755
C06200=1182.891,109.360,-51.844,-178.794,6.166,148.754
C06201=1182.886,109.611,-51.863,-178.792,6.166,148.754
C06202=1182.882,109.859,-51.882,-178.789,6.168,148.753
C06203=1182.877,110.109,-51.902,-178.787,6.169,148.753
C06204=1182.872,110.358,-51.920,-178.784,6.171,148.752
C06205=1182.867,110.607,-51.939,-178.781,6.172,148.752
C06206=1182.863,110.856,-51.958,-178.779,6.173,148.751
C06207=1182.857,111.105,-51.977,-178.776,6.175,148.751
C06208=1182.852,111.355,-51.996,-178.773,6.175,148.750
C06209=1182.848,111.604,-52.015,-178.771,6.177,148.750
C06210=1182.843,111.854,-52.034,-178.768,6.179,148.749
C06211=1182.838,112.102,-52.053,-178.765,6.180,148.749
C06212=1182.833,112.352,-52.072,-178.763,6.181,148.749
C06213=1182.829,112.600,-52.091,-178.759,6.183,148.748
C06214=1182.824,112.851,-52.110,-178.757,6.184,148.748
C06215=1182.818,113.099,-52.129,-178.755,6.185,148.747
C06216=1182.814,113.349,-52.148,-178.752,6.186,148.746
C06217=1182.809,113.598,-52.168,-178.749,6.188,148.746
C06218=1182.805,113.847,-52.186,-178.747,6.189,148.746
C06219=1182.799,114.096,-52.205,-178.744,6.190,148.745
C06220=1182.794,114.346,-52.225,-178.741,6.192,148.745
C06221=1182.790,114.594,-52.244,-178.739,6.193,148.744
C06222=1182.785,114.844,-52.263,-178.736,6.194,148.744
C06223=1182.780,115.093,-52.283,-178.733,6.196,148.743
C06224=1182.775,115.343,-52.301,-178.731,6.197,148.743
C06225=1182.770,115.592,-52.320,-178.728,6.198,148.742
C06226=1182.765,115.841,-52.340,-178.725,6.200,148.742
C06227=1182.761,116.090,-52.359,-178.723,6.201,148.741
C06228=1182.756,116.339,-52.378,-178.720,6.202,148.741
C06229=1182.751,116.588,-52.397,-178.717,6.204,148.740
C06230=1182.747,116.837,-52.417,-178.715,6.205,148.740
C06231=1182.741,117.086,-52.436,-178.712,6.206,148.739
C06232=1182.737,117.336,-52.455,-178.709,6.208,148.739
C06233=1182.733,117.585,-52.475,-178.707,6.209,148.738
C06234=1182.727,117.834,-52.494,-178.704,6.210,148.738
C06235=1182.722,118.084,-52.513,-178.701,6.212,148.737
C06236=1182.717,118.332,-52.533,-178.699,6.213,148.737
C06237=1182.713,118.582,-52.552,-178.696,6.214,148.736
C06238=1182.708,118.831,-52.571,-178.693,6.216,148.736
C06239=1182.703,119.080,-52.591,-178.691,6.217,148.736
C06240=1182.698,119.330,-52.610,-178.688,6.219,148.735
C06241=1182.694,119.578,-52.629,-178.685,6.220,148.735
C06242=1182.689,119.828,-52.649,-178.683,6.221,148.734
C06243=1182.684,120.077,-52.668,-178.680,6.223,148.734
C06244=1182.679,120.326,-52.688,-178.677,6.224,148.733
C06245=1182.674,120.576,-52.707,-178.675,6.225,148.733
C06246=1182.670,120.824,-52.726,-178.672,6.227,148.732
C06247=1182.665,121.074,-52.746,-178.669,6.228,148.732
C06248=1182.660,121.324,-52.765,-178.667,6.229,148.731
C06249=1182.655,121.572,-52.785,-178.664,6.231,148.731
C06250=1182.650,121.822,-52.804,-178.662,6.233,148.730
C06251=1182.646,122.071,-52.823,-178.659,6.233,148.730
C06252=1182.641,122.319,-52.843,-178.656,6.235,148.729
C06253=1182.636,122.569,-52.863,-178.654,6.237,148.729
C06254=1182.631,122.818,-52.882,-178.651,6.237,148.728
C06255=1182.626,123.067,-52.902,-178.648,6.239,148.728
C06256=1182.621,123.317,-52.922,-178.646,6.241,148.728
C06257=1182.617,123.567,-52.941,-178.643,6.242,148.727
C06258=1182.612,123.815,-52.961,-178.640,6.243,148.727
C06259=1182.608,124.064,-52.980,-178.638,6.245,148.726
C06260=1182.603,124.314,-53.000,-178.635,6.246,148.726
C06261=1182.597,124.563,-53.019,-178.633,6.247,148.725
C06262=1182.593,124.811,-53.040,-178.630,6.249,148.725
C06263=1182.588,125.061,-53.059,-178.627,6.251,148.724
C06264=1182.583,125.310,-53.079,-178.625,6.251,148.724
C06265=1182.578,125.559,-53.098,-178.622,6.253,148.723
C06266=1182.574,125.808,-53.119,-178.619,6.255,148.723
C06267=1182.569,126.058,-53.138,-178.617,6.256,148.723
C06268=1182.564,126.307,-53.158,-178.614,6.257,148.722
C06269=1182.559,126.556,-53.178,-178.611,6.259,148.722
C06270=1182.555,126.805,-53.198,-178.608,6.260,148.721
C06271=1182.549,127.054,-53.217,-178.606,6.261,148.721
C06272=1182.545,127.303,-53.237,-178.603,6.263,148.720
C06273=1182.540,127.553,-53.257,-178.600,6.264,148.720
C06274=1182.535,127.802,-53.277,-178.598,6.265,148.719
C06275=1182.531,128.051,-53.297,-178.595,6.267,148.719
C06276=1182.525,128.300,-53.316,-178.593,6.269,148.719
C06277=1182.521,128.550,-53.336,-178.589,6.270,148.718
C06278=1182.516,128.799,-53.356,-178.587,6.271,148.718
C06279=1182.512,129.048,-53.376,-178.585,6.273,148.717
C06280=1182.506,129.296,-53.396,-178.582,6.275,148.717
C06281=1182.502,129.546,-53.416,-178.579,6.275,148.716
C06282=1182.497,129.795,-53.436,-178.577,6.277,148.716
C06283=1182.493,130.045,-53.456,-178.574,6.279,148.715
C06284=1182.488,130.294,-53.476,-178.571,6.281,148.715
C06285=1182.483,130.542,-53.495,-178.569,6.281,148.714
C06286=1182.478,130.791,-53.516,-178.566,6.283,148.714
C06287=1182.474,131.041,-53.535,-178.563,6.285,148.714
C06288=1182.469,131.290,-53.556,-178.561,6.286,148.713
C06289=1182.464,131.539,-53.575,-178.558,6.287,148.712
C06290=1182.459,131.788,-53.596,-178.555,6.289,148.712
C06291=1182.454,132.038,-53.616,-178.553,6.290,148.712
C06292=1182.449,132.306,-53.637,-178.550,6.292,148.711
C06293=1182.444,132.575,-53.659,-178.547,6.294,148.711
C06294=1182.439,132.843,-53.680,-178.544,6.295,148.710
C06295=1182.433,133.112,-53.703,-178.541,6.297,148.710
C06296=1182.429,133.361,-53.722,-178.538,6.299,148.709
C06297=1182.424,133.610,-53.743,-178.536,6.299,148.709
C06298=1182.419,133.860,-53.762,-178.533,6.301,148.709
C06299=1182.415,134.109,-53.783,-178.531,6.303,148.708
C06300=1182.410,134.358,-53.804,-178.527,6.304,148.708
C06301=1182.405,134.607,-53.823,-178.525,6.305,148.707
C06302=1182.400,134.856,-53.843,-178.523,6.307,148.707
C06303=1182.396,135.105,-53.864,-178.520,6.309,148.706
C06304=1182.391,135.354,-53.883,-178.517,6.310,148.706
C06305=1182.386,135.603,-53.904,-178.515,6.311,148.705
C06306=1182.381,135.852,-53.925,-178.512,6.313,148.705
C06307=1182.377,136.102,-53.944,-178.509,6.315,148.705
C06308=1182.372,136.351,-53.965,-178.506,6.316,148.704
C06309=1182.367,136.600,-53.986,-178.503,6.318,148.704
C06310=1182.362,136.849,-54.006,-178.501,6.319,148.703
C06311=1182.357,137.098,-54.025,-178.499,6.320,148.703
C06312=1182.353,137.347,-54.046,-178.496,6.322,148.702
C06313=1182.348,137.596,-54.067,-178.493,6.324,148.702
C06314=1182.343,137.845,-54.087,-178.491,6.325,148.701
C06315=1182.339,138.094,-54.107,-178.488,6.326,148.701
C06316=1182.333,138.344,-54.128,-178.485,6.328,148.701
C06317=1182.329,138.593,-54.148,-178.482,6.330,148.700
C06318=1182.324,138.842,-54.168,-178.480,6.332,148.700
C06319=1182.319,139.091,-54.189,-178.478,6.333,148.699
C06320=1182.315,139.340,-54.210,-178.474,6.334,148.699
C06321=1182.310,139.589,-54.230,-178.472,6.336,148.698
C06322=1182.305,139.839,-54.250,-178.469,6.337,148.698
C06323=1182.300,140.088,-54.271,-178.466,6.339,148.698
C06324=1182.296,140.337,-54.291,-178.464,6.340,148.697
C06325=1182.291,140.586,-54.312,-178.461,6.342,148.697
C06326=1182.286,140.835,-54.332,-178.458,6.343,148.696
C06327=1182.282,141.084,-54.353,-178.456,6.345,148.696
C06328=1182.277,141.333,-54.374,-178.453,6.347,148.695
C06329=1182.272,141.582,-54.394,-178.451,6.348,148.695
C06330=1182.267,141.831,-54.415,-178.448,6.349,148.695
C06331=1182.263,142.080,-54.436,-178.445,6.351,148.694
C06332=1182.258,142.329,-54.456,-178.442,6.353,148.694
C06333=1182.253,142.579,-54.477,-178.440,6.354,148.693
C06334=1182.249,142.828,-54.497,-178.437,6.356,148.693
C06335=1182.243,143.077,-54.518,-178.435,6.357,148.693
C06336=1182.239,143.326,-54.539,-178.432,6.359,148.692
C06337=1182.235,143.575,-54.559,-178.429,6.360,148.692
C06338=1182.229,143.824,-54.580,-178.426,6.362,148.691
C06339=1182.225,144.073,-54.600,-178.424,6.364,148.691
C06340=1182.220,144.322,-54.621,-178.421,6.365,148.690
C06341=1182.215,144.571,-54.642,-178.419,6.366,148.690
C06342=1182.210,144.820,-54.663,-178.416,6.368,148.690
C06343=1182.206,145.069,-54.683,-178.413,6.370,148.689
C06344=1182.201,145.319,-54.704,-178.410,6.371,148.689
C06345=1182.197,145.568,-54.725,-178.408,6.373,148.688
C06346=1182.192,145.817,-54.746,-178.405,6.375,148.688
C06347=1182.187,146.066,-54.767,-178.403,6.376,148.687
C06348=1182.182,146.315,-54.788,-178.400,6.378,148.687
C06349=1182.178,146.564,-54.808,-178.397,6.379,148.687
C06350=1182.173,146.813,-54.829,-178.395,6.381,148.686
C06351=1182.167,147.063,-54.850,-178.391,6.383,148.686
C06352=1182.163,147.311,-54.871,-178.389,6.384,148.685
C06353=1182.158,147.560,-54.892,-178.387,6.385,148.685
C06354=1182.154,147.810,-54.913,-178.384,6.387,148.685
C06355=1182.149,148.059,-54.934,-178.381,6.389,148.684
C06356=1182.145,148.308,-54.954,-178.379,6.391,148.684
C06357=1182.140,148.557,-54.976,-178.376,6.392,148.683
C06358=1182.135,148.806,-54.997,-178.373,6.394,148.683
C06359=1182.130,149.055,-55.017,-178.370,6.395,148.682
C06360=1182.125,149.304,-55.038,-178.368,6.396,148.682
C06361=1182.121,149.552,-55.059,-178.365,6.398,148.682
C06362=1182.116,149.802,-55.081,-178.363,6.400,148.681
C06363=1182.111,150.052,-55.101,-178.360,6.402,148.681
C06364=1182.107,150.300,-55.123,-178.357,6.403,148.681
C06365=1182.102,150.549,-55.144,-178.354,6.405,148.680
C06366=1182.097,150.798,-55.165,-178.352,6.407,148.680
C06367=1182.093,151.047,-55.186,-178.349,6.409,148.679
C06368=1182.088,151.297,-55.207,-178.347,6.409,148.679
C06369=1182.083,151.546,-55.228,-178.344,6.411,148.678
C06370=1182.079,151.794,-55.249,-178.341,6.413,148.678
C06371=1182.073,152.044,-55.270,-178.338,6.415,148.678
C06372=1182.069,152.292,-55.292,-178.336,6.416,148.677
C06373=1182.064,152.542,-55.313,-178.333,6.418,148.677
C06374=1182.060,152.791,-55.333,-178.330,6.420,148.676
C06375=1182.055,153.040,-55.355,-178.328,6.422,148.676
C06376=1182.050,153.289,-55.376,-178.325,6.423,148.676
C06377=1182.045,153.538,-55.398,-178.323,6.424,148.675
C06378=1182.041,153.787,-55.418,-178.320,6.426,148.675
C06379=1182.036,154.036,-55.440,-178.317,6.428,148.674
C06380=1182.031,154.285,-55.461,-178.314,6.429,148.674
C06381=1182.026,154.534,-55.483,-178.312,6.431,148.674
C06382=1182.022,154.784,-55.503,-178.309,6.433,148.673
C06383=1182.017,155.032,-55.525,-178.306,6.435,148.673
C06384=1182.012,155.281,-55.546,-178.304,6.436,148.672
C06385=1182.007,155.530,-55.568,-178.301,6.438,148.672
C06386=1182.003,155.780,-55.589,-178.298,6.440,148.672
C06387=1181.998,156.028,-55.610,-178.296,6.441,148.671
C06388=1181.994,156.277,-55.632,-178.293,6.443,148.671
C06389=1181.989,156.527,-55.653,-178.291,6.444,148.671
C06390=1181.984,156.776,-55.675,-178.288,6.446,148.670
C06391=1181.979,157.025,-55.696,-178.285,6.448,148.670
C06392=1181.974,157.274,-55.718,-178.282,6.449,148.669
C06393=1181.971,157.523,-55.739,-178.280,6.451,148.669
C06394=1181.965,157.772,-55.760,-178.277,6.453,148.668
C06395=1181.961,158.020,-55.782,-178.274,6.455,148.668
C06396=1181.955,158.290,-55.805,-178.271,6.456,148.668
C06397=1181.950,158.559,-55.828,-178.269,6.458,148.667
C06398=1181.945,158.828,-55.852,-178.266,6.460,148.667
C06399=1181.940,159.097,-55.875,-178.263,6.461,148.666
C06400=1181.936,159.345,-55.896,-178.260,6.463,148.666
C06401=1181.931,159.595,-55.918,-178.258,6.465,148.666
C06402=1181.926,159.844,-55.939,-178.255,6.467,148.665
C06403=1181.921,160.093,-55.961,-178.252,6.468,148.665
C06404=1181.917,160.342,-55.983,-178.250,6.470,148.665
C06405=1181.912,160.591,-56.004,-178.247,6.472,148.664
C06406=1181.907,160.840,-56.026,-178.244,6.474,148.664
C06407=1181.903,161.089,-56.048,-178.241,6.476,148.663
C06408=1181.898,161.338,-56.069,-178.239,6.477,148.663
C06409=1181.893,161.587,-56.091,-178.236,6.479,148.663
C06410=1181.888,161.836,-56.112,-178.233,6.481,148.662
C06411=1181.883,162.085,-56.134,-178.231,6.483,148.662
C06412=1181.879,162.334,-56.156,-178.228,6.484,148.662
C06413=1181.874,162.583,-56.178,-178.225,6.486,148.661
C06414=1181.870,162.832,-56.200,-178.223,6.488,148.661
C06415=1181.865,163.081,-56.222,-178.220,6.490,148.660
C06416=1181.860,163.330,-56.243,-178.217,6.491,148.660
C06417=1181.856,163.580,-56.265,-178.215,6.493,148.660
C06418=1181.851,163.828,-56.286,-178.212,6.495,148.659
C06419=1181.847,164.078,-56.308,-178.210,6.496,148.659
C06420=1181.842,164.326,-56.330,-178.207,6.498,148.659
C06421=1181.837,164.575,-56.352,-178.204,6.500,148.658
C06422=1181.833,164.824,-56.374,-178.202,6.501,148.658
C06423=1181.828,165.073,-56.395,-178.199,6.503,148.657
C06424=1181.823,165.322,-56.417,-178.196,6.504,148.657
C06425=1181.819,165.571,-56.439,-178.193,6.506,148.657
C06426=1181.814,165.820,-56.461,-178.191,6.508,148.656
C06427=1181.809,166.069,-56.483,-178.188,6.510,148.656
C06428=1181.804,166.318,-56.506,-178.185,6.512,148.655
C06429=1181.800,166.567,-56.527,-178.183,6.513,148.655
C06430=1181.795,166.816,-56.549,-178.180,6.515,148.655
C06431=1181.790,167.065,-56.571,-178.177,6.517,148.654
C06432=1181.786,167.314,-56.593,-178.175,6.519,148.654
C06433=1181.781,167.563,-56.615,-178.172,6.520,148.654
C06434=1181.777,167.812,-56.637,-178.169,6.522,148.653
C06435=1181.772,168.061,-56.660,-178.166,6.524,148.653
C06436=1181.767,168.310,-56.682,-178.164,6.526,148.652
C06437=1181.763,168.559,-56.703,-178.161,6.528,148.652
C06438=1181.758,168.808,-56.726,-178.159,6.530,148.652
C06439=1181.753,169.057,-56.747,-178.156,6.531,148.652
C06440=1181.748,169.306,-56.770,-178.154,6.533,148.651
C06441=1181.744,169.555,-56.792,-178.151,6.535,148.651
C06442=1181.739,169.804,-56.814,-178.148,6.537,148.650
C06443=1181.735,170.052,-56.836,-178.146,6.539,148.650
C06444=1181.730,170.302,-56.859,-178.143,6.540,148.650
C06445=1181.725,170.551,-56.880,-178.140,6.542,148.649
C06446=1181.721,170.800,-56.902,-178.137,6.544,148.649
C06447=1181.716,171.049,-56.924,-178.135,6.546,148.649
C06448=1181.711,171.298,-56.947,-178.132,6.547,148.648
C06449=1181.706,171.546,-56.969,-178.129,6.549,148.648
C06450=1181.702,171.796,-56.991,-178.127,6.551,148.648
C06451=1181.697,172.045,-57.014,-178.124,6.553,148.647
C06452=1181.692,172.293,-57.036,-178.121,6.554,148.647
C06453=1181.688,172.543,-57.058,-178.119,6.556,148.646
C06454=1181.683,172.791,-57.080,-178.116,6.558,148.646
C06455=1181.678,173.040,-57.103,-178.113,6.560,148.646
C06456=1181.674,173.289,-57.125,-178.111,6.562,148.645
C06457=1181.669,173.538,-57.147,-178.107,6.564,148.645
C06458=1181.665,173.787,-57.170,-178.105,6.566,148.645
C06459=1181.660,174.036,-57.192,-178.102,6.568,148.644
C06460=1181.655,174.286,-57.215,-178.099,6.570,148.644
C06461=1181.651,174.534,-57.237,-178.097,6.571,148.644
C06462=1181.646,174.783,-57.259,-178.094,6.573,148.643
C06463=1181.641,175.032,-57.282,-178.091,6.575,148.643
C06464=1181.636,175.281,-57.304,-178.089,6.577,148.642
C06465=1181.632,175.530,-57.326,-178.087,6.579,148.642
C06466=1181.627,175.779,-57.350,-178.084,6.581,148.642
C06467=1181.623,176.028,-57.371,-178.081,6.582,148.642
C06468=1181.618,176.277,-57.395,-178.078,6.584,148.641
C06469=1181.614,176.526,-57.417,-178.076,6.586,148.641
C06470=1181.608,176.774,-57.440,-178.073,6.588,148.641
C06471=1181.604,177.024,-57.462,-178.070,6.589,148.640
C06472=1181.600,177.272,-57.484,-178.068,6.591,148.640
C06473=1181.594,177.521,-57.507,-178.065,6.593,148.639
C06474=1181.590,177.770,-57.529,-178.062,6.595,148.639
C06475=1181.585,178.020,-57.552,-178.060,6.597,148.639
C06476=1181.581,178.268,-57.575,-178.057,6.598,148.638
C06477=1181.576,178.517,-57.597,-178.054,6.601,148.638
C06478=1181.572,178.766,-57.620,-178.051,6.603,148.638
C06479=1181.567,179.015,-57.643,-178.049,6.605,148.638
C06480=1181.562,179.264,-57.665,-178.046,6.607,148.637
C06481=1181.558,179.513,-57.688,-178.044,6.608,148.637
C06482=1181.553,179.762,-57.710,-178.041,6.610,148.636
C06483=1181.548,180.010,-57.733,-178.038,6.612,148.636
C06484=1181.544,180.259,-57.756,-178.036,6.614,148.636
C06485=1181.539,180.509,-57.779,-178.033,6.616,148.635
C06486=1181.535,180.758,-57.802,-178.030,6.617,148.635
C06487=1181.530,181.006,-57.825,-178.028,6.619,148.635
C06488=1181.525,181.256,-57.847,-178.025,6.621,148.634
C06489=1181.521,181.504,-57.870,-178.022,6.623,148.634
C06490=1181.516,181.753,-57.893,-178.019,6.626,148.634
C06491=1181.512,182.001,-57.916,-178.017,6.627,148.633
C06492=1181.507,182.251,-57.938,-178.014,6.629,148.633
C06493=1181.502,182.500,-57.962,-178.011,6.631,148.633
C06494=1181.498,182.749,-57.984,-178.009,6.633,148.632
C06495=1181.493,182.998,-58.008,-178.006,6.635,148.632
C06496=1181.488,183.246,-58.030,-178.003,6.636,148.632
C06497=1181.484,183.495,-58.053,-178.001,6.638,148.631
C06498=1181.479,183.744,-58.076,-177.999,6.640,148.631
C06499=1181.475,183.993,-58.099,-177.996,6.642,148.631
C06500=1181.470,184.263,-58.124,-177.993,6.645,148.630
C06501=1181.464,184.533,-58.149,-177.990,6.646,148.630
C06502=1181.460,184.802,-58.174,-177.987,6.649,148.630
C06503=1181.454,185.072,-58.199,-177.984,6.651,148.629
C06504=1181.450,185.321,-58.222,-177.981,6.653,148.629
C06505=1181.445,185.569,-58.244,-177.979,6.654,148.629
C06506=1181.441,185.818,-58.268,-177.976,6.656,148.628
C06507=1181.436,186.067,-58.291,-177.973,6.658,148.628
C06508=1181.432,186.316,-58.314,-177.970,6.660,148.628
C06509=1181.427,186.565,-58.337,-177.967,6.662,148.627
C06510=1181.422,186.814,-58.360,-177.965,6.664,148.627
C06511=1181.417,187.063,-58.383,-177.963,6.666,148.627
C06512=1181.413,187.312,-58.406,-177.960,6.668,148.626
C06513=1181.408,187.561,-58.429,-177.957,6.670,148.626
C06514=1181.403,187.810,-58.452,-177.955,6.672,148.626
C06515=1181.399,188.059,-58.476,-177.952,6.673,148.625
C06516=1181.395,188.307,-58.498,-177.949,6.676,148.625
C06517=1181.390,188.556,-58.522,-177.946,6.678,148.625
C06518=1181.385,188.805,-58.545,-177.944,6.680,148.625
C06519=1181.381,189.054,-58.568,-177.941,6.682,148.624
C06520=1181.375,189.303,-58.591,-177.938,6.683,148.624
C06521=1181.371,189.551,-58.616,-177.936,6.685,148.624
C06522=1181.367,189.800,-58.638,-177.933,6.687,148.623
C06523=1181.362,190.049,-58.662,-177.930,6.690,148.623
C06524=1181.358,190.298,-58.685,-177.928,6.692,148.623
C06525=1181.353,190.547,-58.708,-177.925,6.694,148.622
C06526=1181.348,190.796,-58.732,-177.922,6.695,148.622
C06527=1181.344,191.045,-58.755,-177.920,6.697,148.622
C06528=1181.339,191.294,-58.778,-177.917,6.699,148.621
C06529=1181.335,191.543,-58.801,-177.915,6.701,148.621
C06530=1181.331,191.791,-58.825,-177.912,6.704,148.621
C06531=1181.326,192.040,-58.849,-177.909,6.705,148.621
C06532=1181.321,192.289,-58.872,-177.906,6.707,148.620
C06533=1181.316,192.538,-58.895,-177.904,6.709,148.620
C06534=1181.312,192.787,-58.919,-177.901,6.711,148.619
C06535=1181.307,193.035,-58.942,-177.899,6.713,148.619
C06536=1181.302,193.284,-58.966,-177.895,6.716,148.619
C06537=1181.297,193.533,-58.989,-177.893,6.717,148.619
C06538=1181.293,193.782,-59.012,-177.890,6.719,148.618
C06539=1181.288,194.031,-59.037,-177.887,6.721,148.618
C06540=1181.284,194.280,-59.060,-177.885,6.723,148.618
C06541=1181.279,194.529,-59.083,-177.883,6.725,148.617
C06542=1181.274,194.777,-59.107,-177.879,6.727,148.617
C06543=1181.270,195.026,-59.131,-177.877,6.729,148.617
C06544=1181.265,195.275,-59.154,-177.874,6.731,148.616
C06545=1181.260,195.524,-59.177,-177.872,6.733,148.616
C06546=1181.257,195.773,-59.202,-177.869,6.735,148.616
C06547=1181.252,196.022,-59.225,-177.866,6.738,148.616
C06548=1181.247,196.271,-59.249,-177.863,6.739,148.615
C06549=1181.243,196.520,-59.273,-177.861,6.741,148.615
C06550=1181.238,196.769,-59.296,-177.858,6.743,148.615
C06551=1181.234,197.017,-59.320,-177.856,6.745,148.614
C06552=1181.229,197.266,-59.343,-177.853,6.748,148.614
C06553=1181.225,197.515,-59.368,-177.850,6.749,148.614
C06554=1181.220,197.764,-59.391,-177.848,6.752,148.614
C06555=1181.215,198.012,-59.415,-177.845,6.753,148.613
C06556=1181.211,198.261,-59.438,-177.842,6.755,148.613
C06557=1181.206,198.510,-59.462,-177.839,6.758,148.613
C06558=1181.201,198.759,-59.486,-177.836,6.760,148.612
C06559=1181.196,199.008,-59.510,-177.834,6.762,148.612
C06560=1181.192,199.256,-59.534,-177.832,6.763,148.612
C06561=1181.188,199.506,-59.558,-177.829,6.765,148.611
C06562=1181.183,199.754,-59.582,-177.826,6.768,148.611
C06563=1181.179,200.003,-59.606,-177.823,6.770,148.611
C06564=1181.174,200.252,-59.629,-177.821,6.772,148.611
C06565=1181.170,200.500,-59.653,-177.818,6.774,148.610
C06566=1181.164,200.750,-59.677,-177.815,6.776,148.610
C06567=1181.160,200.998,-59.701,-177.813,6.778,148.610
C06568=1181.155,201.247,-59.724,-177.810,6.780,148.610
C06569=1181.152,201.496,-59.749,-177.807,6.782,148.609
C06570=1181.147,201.745,-59.773,-177.805,6.784,148.609
C06571=1181.142,201.994,-59.797,-177.802,6.787,148.609
C06572=1181.137,202.242,-59.821,-177.799,6.788,148.608
C06573=1181.133,202.491,-59.845,-177.797,6.790,148.608
C06574=1181.128,202.740,-59.868,-177.794,6.792,148.608
C06575=1181.124,202.988,-59.893,-177.791,6.795,148.608
C06576=1181.119,203.238,-59.918,-177.789,6.797,148.607
C06577=1181.115,203.487,-59.941,-177.786,6.799,148.607
C06578=1181.110,203.735,-59.965,-177.783,6.800,148.607
C06579=1181.106,203.984,-59.989,-177.780,6.803,148.607
C06580=1181.101,204.232,-60.014,-177.778,6.805,148.606
C06581=1181.097,204.482,-60.037,-177.775,6.807,148.606
C06582=1181.092,204.730,-60.062,-177.773,6.809,148.606
C06583=1181.087,204.979,-60.086,-177.770,6.812,148.605
C06584=1181.083,205.228,-60.110,-177.767,6.813,148.605
C06585=1181.078,205.476,-60.134,-177.764,6.815,148.605
C06586=1181.073,205.726,-60.159,-177.762,6.817,148.605
C06587=1181.069,205.974,-60.183,-177.759,6.820,148.604
C06588=1181.065,206.223,-60.207,-177.756,6.822,148.604
C06589=1181.060,206.472,-60.232,-177.754,6.824,148.604
C06590=1181.056,206.721,-60.256,-177.751,6.826,148.603
C06591=1181.051,206.969,-60.280,-177.748,6.828,148.603
C06592=1181.046,207.218,-60.305,-177.746,6.830,148.603
C06593=1181.041,207.467,-60.328,-177.743,6.832,148.603
C06594=1181.037,207.716,-60.353,-177.741,6.834,148.602
C06595=1181.033,207.965,-60.377,-177.738,6.837,148.602
C06596=1181.028,208.213,-60.401,-177.735,6.839,148.602
C06597=1181.023,208.462,-60.426,-177.733,6.841,148.602
C06598=1181.019,208.711,-60.450,-177.729,6.843,148.601
C06599=1181.014,208.960,-60.475,-177.727,6.845,148.601
C06600=1181.010,209.208,-60.499,-177.725,6.847,148.601
C06601=1181.005,209.457,-60.524,-177.722,6.849,148.600
C06602=1181.001,209.706,-60.548,-177.719,6.852,148.600
C06603=1180.996,209.954,-60.572,-177.717,6.854,148.600
C06604=1180.991,210.224,-60.599,-177.713,6.856,148.600
C06605=1180.987,210.495,-60.626,-177.711,6.858,148.599
C06606=1180.982,210.766,-60.653,-177.707,6.861,148.599
C06607=1180.976,211.036,-60.679,-177.705,6.863,148.599
C06608=1180.972,211.286,-60.704,-177.702,6.866,148.599
C06609=1180.967,211.534,-60.729,-177.699,6.867,148.598
C06610=1180.962,211.782,-60.753,-177.697,6.869,148.598
C06611=1180.959,212.031,-60.778,-177.694,6.871,148.598
C06612=1180.953,212.280,-60.802,-177.691,6.874,148.598
C06613=1180.949,212.528,-60.826,-177.689,6.876,148.597
C06614=1180.944,212.778,-60.851,-177.686,6.878,148.597
C06615=1180.940,213.026,-60.876,-177.683,6.880,148.597
C06616=1180.935,213.274,-60.901,-177.681,6.882,148.596
C06617=1180.931,213.524,-60.925,-177.678,6.884,148.596
C06618=1180.926,213.772,-60.950,-177.675,6.887,148.596
C06619=1180.922,214.022,-60.975,-177.673,6.889,148.596
C06620=1180.917,214.270,-60.999,-177.670,6.891,148.596
C06621=1180.913,214.518,-61.025,-177.667,6.894,148.595
C06622=1180.909,214.767,-61.049,-177.665,6.896,148.595
C06623=1180.904,215.016,-61.074,-177.662,6.898,148.595
C06624=1180.899,215.265,-61.099,-177.659,6.900,148.594
C06625=1180.895,215.513,-61.123,-177.657,6.902,148.594
C06626=1180.890,215.762,-61.148,-177.654,6.904,148.594
C06627=1180.885,216.011,-61.173,-177.651,6.907,148.594
C06628=1180.881,216.259,-61.198,-177.649,6.909,148.594
C06629=1180.877,216.509,-61.223,-177.646,6.911,148.593
C06630=1180.872,216.757,-61.248,-177.643,6.913,148.593
C06631=1180.868,217.006,-61.273,-177.641,6.915,148.593
C06632=1180.863,217.255,-61.298,-177.638,6.917,148.593
C06633=1180.858,217.503,-61.322,-177.635,6.920,148.592
C06634=1180.854,217.752,-61.347,-177.633,6.922,148.592
C06635=1180.849,218.001,-61.372,-177.630,6.924,148.592
C06636=1180.845,218.250,-61.397,-177.627,6.927,148.592
C06637=1180.841,218.498,-61.422,-177.625,6.929,148.591
C06638=1180.836,218.747,-61.447,-177.622,6.931,148.591
C06639=1180.831,218.995,-61.472,-177.619,6.933,148.591
C06640=1180.827,219.245,-61.497,-177.616,6.935,148.591
C06641=1180.823,219.492,-61.522,-177.614,6.937,148.590
C06642=1180.818,219.742,-61.547,-177.611,6.940,148.590
C06643=1180.813,219.990,-61.572,-177.608,6.942,148.590
C06644=1180.809,220.239,-61.598,-177.606,6.944,148.590
C06645=1180.804,220.488,-61.623,-177.603,6.946,148.589
C06646=1180.800,220.737,-61.647,-177.601,6.949,148.589
C06647=1180.795,220.985,-61.673,-177.598,6.950,148.589
C06648=1180.791,221.234,-61.698,-177.595,6.953,148.589
C06649=1180.786,221.482,-61.723,-177.593,6.955,148.589
C06650=1180.781,221.732,-61.748,-177.590,6.958,148.588
C06651=1180.778,221.980,-61.773,-177.587,6.960,148.588
C06652=1180.773,222.228,-61.799,-177.585,6.962,148.588
C06653=1180.769,222.478,-61.824,-177.582,6.965,148.588
C06654=1180.764,222.726,-61.849,-177.579,6.967,148.587
C06655=1180.760,222.975,-61.875,-177.577,6.968,148.587
C06656=1180.754,223.223,-61.900,-177.574,6.971,148.587
C06657=1180.750,223.472,-61.925,-177.571,6.973,148.587
C06658=1180.745,223.720,-61.951,-177.569,6.975,148.587
C06659=1180.742,223.969,-61.975,-177.566,6.978,148.586
C06660=1180.737,224.218,-62.001,-177.564,6.980,148.586
C06661=1180.733,224.466,-62.026,-177.560,6.983,148.586
C06662=1180.728,224.716,-62.051,-177.558,6.984,148.585
C06663=1180.723,224.964,-62.077,-177.556,6.987,148.585
C06664=1180.719,225.213,-62.102,-177.552,6.989,148.585
C06665=1180.715,225.461,-62.128,-177.550,6.991,148.585
C06666=1180.710,225.710,-62.153,-177.547,6.994,148.585
C06667=1180.705,225.959,-62.179,-177.545,6.996,148.585
C06668=1180.701,226.207,-62.204,-177.542,6.998,148.584
C06669=1180.696,226.456,-62.230,-177.539,7.001,148.584
C06670=1180.692,226.705,-62.256,-177.537,7.003,148.584
C06671=1180.687,226.953,-62.280,-177.534,7.006,148.584
C06672=1180.683,227.202,-62.306,-177.531,7.008,148.583
C06673=1180.679,227.451,-62.332,-177.529,7.009,148.583
C06674=1180.674,227.699,-62.357,-177.526,7.012,148.583
C06675=1180.669,227.948,-62.383,-177.523,7.014,148.583
C06676=1180.665,228.197,-62.409,-177.521,7.017,148.583
C06677=1180.660,228.445,-62.434,-177.518,7.019,148.582
C06678=1180.656,228.694,-62.460,-177.516,7.021,148.582
C06679=1180.652,228.943,-62.485,-177.512,7.024,148.582
C06680=1180.647,229.191,-62.510,-177.510,7.026,148.582
C06681=1180.643,229.440,-62.536,-177.507,7.028,148.581
C06682=1180.638,229.689,-62.562,-177.505,7.031,148.581
C06683=1180.633,229.937,-62.588,-177.502,7.033,148.581
C06684=1180.629,230.186,-62.613,-177.500,7.035,148.581
C06685=1180.624,230.435,-62.639,-177.497,7.037,148.581
C06686=1180.620,230.684,-62.665,-177.494,7.040,148.581
C06687=1180.615,230.932,-62.690,-177.491,7.042,148.580
C06688=1180.611,231.180,-62.716,-177.489,7.045,148.580
C06689=1180.607,231.429,-62.742,-177.486,7.047,148.580
C06690=1180.602,231.677,-62.767,-177.483,7.050,148.580
C06691=1180.597,231.927,-62.793,-177.481,7.051,148.579
C06692=1180.593,232.175,-62.820,-177.478,7.054,148.579
C06693=1180.589,232.424,-62.846,-177.475,7.056,148.579
C06694=1180.584,232.672,-62.871,-177.473,7.058,148.579
C06695=1180.580,232.920,-62.897,-177.470,7.061,148.579
C06696=1180.576,233.169,-62.923,-177.468,7.063,148.579
C06697=1180.571,233.418,-62.949,-177.464,7.066,148.578
C06698=1180.566,233.666,-62.974,-177.462,7.068,148.578
C06699=1180.562,233.915,-63.000,-177.460,7.071,148.578
C06700=1180.558,234.163,-63.027,-177.457,7.073,148.578
C06701=1180.553,234.413,-63.053,-177.455,7.075,148.578
C06702=1180.549,234.661,-63.079,-177.452,7.078,148.577
C06703=1180.544,234.909,-63.104,-177.449,7.080,148.577
C06704=1180.540,235.158,-63.130,-177.446,7.082,148.577
C06705=1180.535,235.407,-63.157,-177.444,7.084,148.577
C06706=1180.531,235.656,-63.183,-177.441,7.087,148.577
C06707=1180.526,235.904,-63.208,-177.439,7.089,148.576
C06708=1180.521,236.175,-63.237,-177.435,7.092,148.576
C06709=1180.516,236.447,-63.265,-177.433,7.095,148.576
C06710=1180.512,236.718,-63.294,-177.429,7.097,148.576
C06711=1180.507,236.990,-63.322,-177.427,7.100,148.576
C06712=1180.502,237.239,-63.349,-177.424,7.102,148.575
C06713=1180.498,237.488,-63.375,-177.422,7.104,148.575
C06714=1180.493,237.736,-63.400,-177.419,7.107,148.575
C06715=1180.489,237.984,-63.427,-177.416,7.109,148.575
C06716=1180.484,238.233,-63.453,-177.414,7.112,148.575
C06717=1180.480,238.482,-63.479,-177.411,7.114,148.575
C06718=1180.475,238.730,-63.506,-177.408,7.117,148.574
C06719=1180.471,238.979,-63.532,-177.406,7.119,148.574
C06720=1180.467,239.228,-63.559,-177.403,7.122,148.574
C06721=1180.462,239.476,-63.585,-177.400,7.124,148.574
C06722=1180.457,239.725,-63.610,-177.398,7.126,148.574
C06723=1180.453,239.973,-63.637,-177.395,7.129,148.574
C06724=1180.449,240.222,-63.663,-177.392,7.131,148.573
C06725=1180.444,240.470,-63.690,-177.390,7.133,148.573
C06726=1180.440,240.719,-63.716,-177.387,7.136,148.573
C06727=1180.435,240.968,-63.743,-177.385,7.138,148.573
C06728=1180.431,241.216,-63.768,-177.382,7.141,148.573
C06729=1180.426,241.465,-63.795,-177.379,7.143,148.572
C06730=1180.422,241.713,-63.822,-177.376,7.146,148.572
C06731=1180.417,241.962,-63.848,-177.374,7.148,148.572
C06732=1180.413,242.210,-63.875,-177.371,7.151,148.572
C06733=1180.408,242.460,-63.901,-177.369,7.153,148.572
C06734=1180.404,242.708,-63.928,-177.366,7.156,148.572
C06735=1180.399,242.956,-63.954,-177.363,7.158,148.571
C06736=1180.395,243.204,-63.980,-177.361,7.161,148.571
C06737=1180.390,243.453,-64.007,-177.358,7.162,148.571
C06738=1180.386,243.702,-64.033,-177.355,7.165,148.571
C06739=1180.381,243.950,-64.060,-177.353,7.168,148.571
C06740=1180.378,244.198,-64.086,-177.350,7.170,148.571
C06741=1180.373,244.447,-64.113,-177.348,7.172,148.571
C06742=1180.369,244.696,-64.139,-177.345,7.175,148.570
C06743=1180.364,244.944,-64.166,-177.342,7.177,148.570
C06744=1180.359,245.193,-64.193,-177.340,7.180,148.570
C06745=1180.355,245.441,-64.219,-177.337,7.182,148.570
C06746=1180.350,245.690,-64.246,-177.334,7.185,148.570
C06747=1180.347,245.938,-64.273,-177.332,7.187,148.570
C06748=1180.342,246.187,-64.300,-177.329,7.190,148.570
C06749=1180.337,246.436,-64.326,-177.326,7.193,148.569
C06750=1180.333,246.684,-64.352,-177.324,7.195,148.569
C06751=1180.328,246.932,-64.379,-177.321,7.198,148.569
C06752=1180.324,247.182,-64.407,-177.319,7.200,148.569
C06753=1180.320,247.430,-64.433,-177.316,7.203,148.569
C06754=1180.315,247.679,-64.460,-177.314,7.205,148.569
C06755=1180.311,247.927,-64.487,-177.310,7.207,148.568
C06756=1180.307,248.176,-64.513,-177.308,7.210,148.568
C06757=1180.302,248.424,-64.540,-177.306,7.213,148.568
C06758=1180.298,248.673,-64.567,-177.302,7.215,148.568
C06759=1180.294,248.921,-64.594,-177.300,7.217,148.568
C06760=1180.289,249.169,-64.621,-177.297,7.220,148.568
C06761=1180.284,249.418,-64.648,-177.295,7.222,148.567
C06762=1180.280,249.666,-64.675,-177.292,7.225,148.567
C06763=1180.276,249.914,-64.701,-177.290,7.227,148.567
C06764=1180.271,250.163,-64.729,-177.287,7.230,148.567
C06765=1180.267,250.412,-64.756,-177.284,7.232,148.567
C06766=1180.262,250.661,-64.783,-177.282,7.235,148.567
C06767=1180.258,250.909,-64.809,-177.279,7.238,148.567
C06768=1180.254,251.157,-64.837,-177.276,7.240,148.566
C06769=1180.249,251.406,-64.864,-177.274,7.243,148.566
C06770=1180.244,251.654,-64.891,-177.271,7.245,148.566
C06771=1180.241,251.902,-64.917,-177.269,7.248,148.566
C06772=1180.236,252.151,-64.944,-177.266,7.250,148.566
C06773=1180.232,252.400,-64.972,-177.263,7.253,148.566
C06774=1180.227,252.649,-64.999,-177.261,7.256,148.566
C06775=1180.223,252.897,-65.026,-177.258,7.257,148.566
C06776=1180.218,253.146,-65.053,-177.255,7.260,148.565
C06777=1180.214,253.394,-65.079,-177.253,7.263,148.565
C06778=1180.210,253.642,-65.107,-177.250,7.266,148.565
C06779=1180.206,253.891,-65.134,-177.247,7.268,148.565
C06780=1180.201,254.139,-65.162,-177.245,7.270,148.565
C06781=1180.196,254.388,-65.189,-177.242,7.273,148.565
C06782=1180.192,254.636,-65.216,-177.240,7.276,148.565
C06783=1180.187,254.885,-65.243,-177.237,7.278,148.565
C06784=1180.183,255.133,-65.271,-177.234,7.281,148.564
C06785=1180.179,255.382,-65.298,-177.232,7.283,148.564
C06786=1180.174,255.630,-65.325,-177.229,7.286,148.564
C06787=1180.169,255.879,-65.352,-177.227,7.288,148.564
C06788=1180.166,256.126,-65.379,-177.224,7.291,148.564
C06789=1180.162,256.376,-65.407,-177.221,7.294,148.564
C06790=1180.157,256.624,-65.434,-177.219,7.296,148.564
C06791=1180.153,256.872,-65.461,-177.216,7.299,148.564
C06792=1180.148,257.121,-65.489,-177.214,7.301,148.563
C06793=1180.144,257.370,-65.516,-177.211,7.304,148.563
C06794=1180.139,257.618,-65.544,-177.208,7.307,148.563
C06795=1180.135,257.866,-65.571,-177.206,7.309,148.563
C06796=1180.130,258.115,-65.598,-177.203,7.312,148.563
C06797=1180.126,258.363,-65.626,-177.200,7.315,148.563
C06798=1180.122,258.612,-65.653,-177.198,7.317,148.563
C06799=1180.117,258.860,-65.680,-177.195,7.320,148.563
C06800=1180.113,259.108,-65.708,-177.193,7.322,148.563
C06801=1180.108,259.358,-65.736,-177.190,7.325,148.563
C06802=1180.104,259.605,-65.764,-177.187,7.328,148.562
C06803=1180.099,259.854,-65.791,-177.185,7.330,148.562
C06804=1180.095,260.103,-65.819,-177.182,7.333,148.562
C06805=1180.091,260.351,-65.846,-177.179,7.336,148.562
C06806=1180.086,260.599,-65.874,-177.177,7.338,148.562
C06807=1180.082,260.848,-65.901,-177.174,7.341,148.562
C06808=1180.078,261.096,-65.929,-177.171,7.344,148.562
C06809=1180.073,261.344,-65.956,-177.169,7.346,148.562
C06810=1180.069,261.592,-65.984,-177.166,7.349,148.562
C06811=1180.065,261.842,-66.011,-177.164,7.351,148.561
C06812=1180.059,262.114,-66.042,-177.161,7.353,148.561
C06813=1180.055,262.387,-66.072,-177.158,7.356,148.561
C06814=1180.050,262.661,-66.103,-177.155,7.359,148.561
C06815=1180.045,262.933,-66.133,-177.152,7.363,148.561
C06816=1180.041,263.182,-66.161,-177.149,7.365,148.561
C06817=1180.037,263.430,-66.189,-177.147,7.368,148.561
C06818=1180.032,263.678,-66.216,-177.145,7.370,148.561
C06819=1180.028,263.927,-66.245,-177.142,7.373,148.561
C06820=1180.023,264.175,-66.273,-177.139,7.376,148.561
C06821=1180.019,264.424,-66.300,-177.137,7.378,148.560
C06822=1180.015,264.672,-66.328,-177.134,7.381,148.560
C06823=1180.010,264.920,-66.356,-177.131,7.384,148.560
C06824=1180.006,265.170,-66.384,-177.129,7.386,148.560
C06825=1180.001,265.417,-66.411,-177.126,7.389,148.560
C06826=1179.997,265.665,-66.439,-177.123,7.392,148.560
C06827=1179.993,265.914,-66.468,-177.121,7.394,148.560
C06828=1179.988,266.162,-66.496,-177.118,7.397,148.560
C06829=1179.984,266.411,-66.523,-177.116,7.400,148.560
C06830=1179.979,266.660,-66.552,-177.113,7.403,148.560
C06831=1179.975,266.908,-66.580,-177.110,7.405,148.559
C06832=1179.971,267.156,-66.607,-177.108,7.408,148.559
C06833=1179.967,267.404,-66.635,-177.105,7.411,148.559
C06834=1179.962,267.653,-66.663,-177.103,7.413,148.559
C06835=1179.957,267.901,-66.691,-177.100,7.416,148.559
C06836=1179.953,268.150,-66.720,-177.097,7.419,148.559
C06837=1179.949,268.398,-66.748,-177.095,7.421,148.559
C06838=1179.945,268.647,-66.776,-177.092,7.424,148.559
C06839=1179.940,268.895,-66.804,-177.090,7.427,148.559
C06840=1179.936,269.143,-66.832,-177.087,7.429,148.559
C06841=1179.932,269.391,-66.860,-177.084,7.432,148.559
C06842=1179.927,269.640,-66.889,-177.081,7.435,148.559
C06843=1179.923,269.888,-66.917,-177.079,7.438,148.559
C06844=1179.918,270.137,-66.945,-177.077,7.440,148.558
C06845=1179.914,270.385,-66.973,-177.074,7.443,148.558
C06846=1179.910,270.633,-67.001,-177.071,7.446,148.558
C06847=1179.905,270.881,-67.030,-177.069,7.448,148.558
C06848=1179.901,271.130,-67.058,-177.066,7.451,148.558
C06849=1179.896,271.378,-67.086,-177.063,7.454,148.558
C06850=1179.893,271.627,-67.114,-177.061,7.456,148.558
C06851=1179.887,271.875,-67.143,-177.059,7.459,148.558
C06852=1179.884,272.124,-67.171,-177.056,7.462,148.558
C06853=1179.879,272.372,-67.199,-177.053,7.465,148.558
C06854=1179.875,272.620,-67.227,-177.050,7.467,148.558
C06855=1179.870,272.869,-67.256,-177.048,7.470,148.558
C06856=1179.866,273.117,-67.284,-177.045,7.473,148.558
C06857=1179.862,273.365,-67.313,-177.043,7.475,148.558
C06858=1179.858,273.613,-67.341,-177.040,7.478,148.557
C06859=1179.853,273.862,-67.370,-177.037,7.481,148.557
C06860=1179.849,274.110,-67.398,-177.035,7.484,148.557
C06861=1179.844,274.359,-67.426,-177.032,7.486,148.557
C06862=1179.841,274.607,-67.455,-177.030,7.489,148.557
C06863=1179.836,274.855,-67.483,-177.027,7.492,148.557
C06864=1179.831,275.104,-67.512,-177.024,7.495,148.557
C06865=1179.827,275.352,-67.540,-177.022,7.497,148.557
C06866=1179.822,275.601,-67.569,-177.019,7.500,148.557
C06867=1179.819,275.849,-67.598,-177.017,7.503,148.557
C06868=1179.814,276.097,-67.626,-177.014,7.506,148.557
C06869=1179.809,276.346,-67.655,-177.012,7.508,148.557
C06870=1179.806,276.594,-67.684,-177.009,7.511,148.557
C06871=1179.801,276.842,-67.712,-177.006,7.514,148.557
C06872=1179.797,277.090,-67.740,-177.004,7.517,148.557
C06873=1179.793,277.339,-67.770,-177.001,7.520,148.557
C06874=1179.788,277.587,-67.798,-176.999,7.523,148.557
C06875=1179.784,277.835,-67.826,-176.996,7.526,148.557
C06876=1179.780,278.084,-67.855,-176.993,7.529,148.557
C06877=1179.775,278.332,-67.884,-176.991,7.531,148.556
C06878=1179.771,278.580,-67.913,-176.988,7.534,148.556
C06879=1179.767,278.829,-67.941,-176.986,7.537,148.556
C06880=1179.762,279.076,-67.971,-176.983,7.540,148.556
C06881=1179.758,279.325,-67.999,-176.981,7.542,148.556
C06882=1179.754,279.574,-68.027,-176.978,7.545,148.556
C06883=1179.749,279.821,-68.057,-176.975,7.548,148.556
C06884=1179.745,280.070,-68.085,-176.973,7.551,148.556
C06885=1179.741,280.318,-68.114,-176.970,7.553,148.556
C06886=1179.737,280.567,-68.143,-176.968,7.556,148.556
C06887=1179.732,280.815,-68.172,-176.965,7.559,148.556
C06888=1179.728,281.063,-68.201,-176.962,7.562,148.556
C06889=1179.724,281.312,-68.230,-176.960,7.564,148.556
C06890=1179.719,281.559,-68.259,-176.957,7.567,148.556
C06891=1179.715,281.808,-68.287,-176.955,7.570,148.556
C06892=1179.710,282.056,-68.317,-176.952,7.573,148.556
C06893=1179.706,282.305,-68.346,-176.949,7.576,148.556
C06894=1179.701,282.553,-68.375,-176.947,7.578,148.556
C06895=1179.698,282.801,-68.403,-176.944,7.581,148.556
C06896=1179.693,283.050,-68.432,-176.941,7.584,148.556
C06897=1179.689,283.298,-68.462,-176.939,7.587,148.556
C06898=1179.684,283.545,-68.491,-176.937,7.589,148.555
C06899=1179.680,283.794,-68.520,-176.934,7.592,148.555
C06900=1179.676,284.043,-68.549,-176.931,7.595,148.555
C06901=1179.671,284.291,-68.578,-176.928,7.598,148.555
C06902=1179.667,284.540,-68.607,-176.926,7.601,148.555
C06903=1179.663,284.787,-68.636,-176.923,7.603,148.555
C06904=1179.659,285.035,-68.665,-176.921,7.606,148.555
C06905=1179.654,285.283,-68.695,-176.918,7.610,148.555
C06906=1179.650,285.532,-68.724,-176.916,7.613,148.555
C06907=1179.646,285.781,-68.753,-176.913,7.616,148.555
C06908=1179.641,286.028,-68.782,-176.911,7.618,148.555
C06909=1179.637,286.276,-68.811,-176.908,7.621,148.555
C06910=1179.633,286.525,-68.841,-176.905,7.624,148.555
C06911=1179.629,286.773,-68.870,-176.903,7.627,148.555
C06912=1179.624,287.022,-68.899,-176.900,7.630,148.555
C06913=1179.620,287.270,-68.928,-176.898,7.632,148.555
C06914=1179.616,287.518,-68.958,-176.895,7.635,148.555
C06915=1179.611,287.766,-68.987,-176.892,7.638,148.555
C06916=1179.607,288.041,-69.019,-176.890,7.641,148.555
C06917=1179.602,288.316,-69.052,-176.887,7.644,148.555
C06918=1179.596,288.590,-69.084,-176.884,7.648,148.555
C06919=1179.593,288.865,-69.117,-176.881,7.651,148.555
C06920=1179.588,289.113,-69.147,-176.878,7.654,148.555
C06921=1179.584,289.361,-69.176,-176.876,7.657,148.555
C06922=1179.579,289.609,-69.205,-176.874,7.659,148.555
C06923=1179.575,289.857,-69.235,-176.871,7.662,148.555
C06924=1179.570,290.106,-69.265,-176.868,7.665,148.555
C06925=1179.566,290.354,-69.294,-176.865,7.668,148.555
C06926=1179.562,290.602,-69.324,-176.863,7.671,148.555
C06927=1179.558,290.851,-69.353,-176.861,7.673,148.555
C06928=1179.554,291.099,-69.383,-176.858,7.676,148.555
C06929=1179.549,291.347,-69.412,-176.855,7.679,148.555
C06930=1179.545,291.595,-69.441,-176.853,7.682,148.555
C06931=1179.541,291.844,-69.471,-176.850,7.685,148.555
C06932=1179.537,292.092,-69.500,-176.847,7.688,148.555
C06933=1179.532,292.341,-69.530,-176.845,7.691,148.555
C06934=1179.528,292.588,-69.561,-176.843,7.694,148.555
C06935=1179.524,292.837,-69.590,-176.840,7.697,148.555
C06936=1179.520,293.085,-69.619,-176.837,7.700,148.555
C06937=1179.516,293.333,-69.649,-176.834,7.703,148.555
C06938=1179.511,293.581,-69.678,-176.832,7.706,148.555
C06939=1179.507,293.829,-69.709,-176.830,7.708,148.555
C06940=1179.503,294.078,-69.739,-176.827,7.711,148.555
C06941=1179.498,294.326,-69.768,-176.824,7.714,148.555
C06942=1179.494,294.574,-69.797,-176.822,7.717,148.555
C06943=1179.490,294.822,-69.828,-176.819,7.720,148.555
C06944=1179.485,295.070,-69.858,-176.817,7.723,148.555
C06945=1179.481,295.319,-69.887,-176.814,7.726,148.555
C06946=1179.477,295.567,-69.917,-176.812,7.728,148.555
C06947=1179.472,295.815,-69.947,-176.809,7.731,148.555
C06948=1179.468,296.063,-69.977,-176.806,7.734,148.555
C06949=1179.464,296.311,-70.006,-176.804,7.737,148.555
C06950=1179.460,296.559,-70.036,-176.801,7.741,148.555
C06951=1179.455,296.808,-70.066,-176.799,7.744,148.555
C06952=1179.451,297.056,-70.096,-176.797,7.746,148.555
C06953=1179.447,297.303,-70.126,-176.794,7.749,148.555
C06954=1179.442,297.552,-70.156,-176.791,7.752,148.555
C06955=1179.438,297.800,-70.186,-176.789,7.755,148.555
C06956=1179.434,298.048,-70.216,-176.786,7.758,148.555
C06957=1179.430,298.296,-70.247,-176.783,7.761,148.555
C06958=1179.425,298.544,-70.276,-176.781,7.764,148.555
C06959=1179.422,298.792,-70.306,-176.778,7.767,148.555
C06960=1179.417,299.041,-70.337,-176.776,7.769,148.555
C06961=1179.413,299.289,-70.366,-176.773,7.773,148.555
C06962=1179.408,299.537,-70.397,-176.771,7.776,148.555
C06963=1179.405,299.785,-70.427,-176.768,7.779,148.555
C06964=1179.400,300.033,-70.456,-176.765,7.782,148.555
C06965=1179.396,300.281,-70.487,-176.763,7.785,148.555
C06966=1179.392,300.529,-70.517,-176.760,7.788,148.555
C06967=1179.387,300.777,-70.547,-176.758,7.791,148.555
C06968=1179.383,301.026,-70.577,-176.755,7.793,148.555
C06969=1179.379,301.274,-70.608,-176.753,7.796,148.555
C06970=1179.375,301.522,-70.638,-176.750,7.799,148.555
C06971=1179.370,301.771,-70.668,-176.748,7.802,148.555
C06972=1179.366,302.018,-70.698,-176.745,7.805,148.555
C06973=1179.361,302.267,-70.728,-176.742,7.808,148.555
C06974=1179.357,302.514,-70.759,-176.740,7.812,148.555
C06975=1179.353,302.763,-70.790,-176.737,7.815,148.555
C06976=1179.349,303.011,-70.820,-176.735,7.817,148.555
C06977=1179.345,303.259,-70.850,-176.732,7.820,148.555
C06978=1179.341,303.507,-70.880,-176.730,7.823,148.555
C06979=1179.336,303.755,-70.911,-176.727,7.826,148.555
C06980=1179.332,304.003,-70.940,-176.725,7.829,148.555
C06981=1179.328,304.252,-70.971,-176.722,7.832,148.555
C06982=1179.324,304.500,-71.002,-176.720,7.835,148.555
C06983=1179.319,304.747,-71.032,-176.717,7.838,148.555
C06984=1179.315,304.995,-71.063,-176.714,7.841,148.555
C06985=1179.311,305.244,-71.093,-176.712,7.844,148.555
C06986=1179.307,305.492,-71.124,-176.710,7.847,148.556
C06987=1179.303,305.740,-71.154,-176.707,7.850,148.556
C06988=1179.298,305.988,-71.185,-176.704,7.853,148.555
C06989=1179.293,306.236,-71.215,-176.702,7.856,148.556
C06990=1179.290,306.484,-71.246,-176.699,7.859,148.556
C06991=1179.285,306.733,-71.276,-176.697,7.862,148.556
C06992=1179.281,306.981,-71.307,-176.694,7.865,148.556
C06993=1179.277,307.228,-71.337,-176.692,7.868,148.556
C06994=1179.273,307.477,-71.368,-176.689,7.871,148.556
C06995=1179.268,307.725,-71.399,-176.686,7.874,148.556
C06996=1179.264,307.973,-71.429,-176.685,7.877,148.556
C06997=1179.260,308.221,-71.460,-176.682,7.880,148.556
C06998=1179.256,308.469,-71.491,-176.679,7.883,148.556
C06999=1179.251,308.717,-71.522,-176.677,7.886,148.556
C07000=1179.247,308.965,-71.552,-176.674,7.889,148.556
C07001=1179.243,309.214,-71.583,-176.671,7.892,148.556
C07002=1179.239,309.462,-71.614,-176.669,7.895,148.556
C07003=1179.235,309.709,-71.644,-176.666,7.898,148.556
C07004=1179.231,309.958,-71.675,-176.664,7.901,148.556
C07005=1179.226,310.206,-71.706,-176.661,7.904,148.556
C07006=1179.221,310.454,-71.737,-176.659,7.908,148.556
C07007=1179.217,310.702,-71.768,-176.656,7.911,148.556
C07008=1179.214,310.949,-71.799,-176.654,7.913,148.556
C07009=1179.209,311.197,-71.829,-176.652,7.916,148.557
C07010=1179.205,311.446,-71.860,-176.649,7.919,148.556
C07011=1179.201,311.694,-71.891,-176.646,7.922,148.556
C07012=1179.196,311.942,-71.922,-176.644,7.925,148.557
C07013=1179.193,312.190,-71.953,-176.641,7.928,148.557
C07014=1179.188,312.438,-71.984,-176.639,7.932,148.557
C07015=1179.184,312.686,-72.015,-176.636,7.935,148.557
C07016=1179.180,312.934,-72.046,-176.633,7.938,148.557
C07017=1179.175,313.182,-72.077,-176.631,7.941,148.557
C07018=1179.171,313.430,-72.107,-176.628,7.944,148.557
C07019=1179.167,313.678,-72.139,-176.626,7.947,148.557
C07020=1179.162,313.955,-72.173,-176.623,7.950,148.557
C07021=1179.158,314.232,-72.208,-176.620,7.954,148.557
C07022=1179.153,314.508,-72.243,-176.617,7.957,148.557
C07023=1179.148,314.784,-72.277,-176.615,7.960,148.557
C07024=1179.144,315.033,-72.309,-176.612,7.963,148.557
C07025=1179.140,315.281,-72.339,-176.610,7.966,148.557
C07026=1179.136,315.529,-72.371,-176.607,7.970,148.558
C07027=1179.132,315.777,-72.402,-176.605,7.973,148.558
C07028=1179.127,316.025,-72.433,-176.602,7.976,148.558
C07029=1179.123,316.273,-72.464,-176.600,7.979,148.558
C07030=1179.119,316.521,-72.495,-176.597,7.982,148.558
C07031=1179.115,316.769,-72.527,-176.595,7.985,148.558
C07032=1179.110,317.017,-72.558,-176.592,7.988,148.558
C07033=1179.106,317.266,-72.589,-176.590,7.992,148.558
C07034=1179.102,317.513,-72.620,-176.587,7.995,148.558
C07035=1179.098,317.762,-72.652,-176.585,7.998,148.558
C07036=1179.094,318.009,-72.683,-176.582,8.001,148.558
C07037=1179.090,318.258,-72.714,-176.579,8.004,148.558
C07038=1179.085,318.505,-72.746,-176.577,8.007,148.559
C07039=1179.081,318.754,-72.777,-176.574,8.010,148.558
C07040=1179.077,319.001,-72.808,-176.573,8.013,148.559
C07041=1179.073,319.249,-72.840,-176.570,8.016,148.559
C07042=1179.069,319.497,-72.871,-176.568,8.019,148.559
C07043=1179.065,319.745,-72.903,-176.565,8.022,148.559
C07044=1179.060,319.993,-72.934,-176.563,8.025,148.559
C07045=1179.057,320.241,-72.965,-176.560,8.028,148.559
C07046=1179.052,320.489,-72.997,-176.557,8.031,148.559
C07047=1179.048,320.737,-73.029,-176.555,8.035,148.559
C07048=1179.043,320.985,-73.060,-176.552,8.038,148.559
C07049=1179.040,321.233,-73.092,-176.550,8.041,148.559
C07050=1179.036,321.481,-73.123,-176.547,8.044,148.559
C07051=1179.031,321.729,-73.154,-176.545,8.047,148.560
C07052=1179.028,321.977,-73.186,-176.542,8.050,148.560
C07053=1179.023,322.225,-73.217,-176.540,8.053,148.560
C07054=1179.018,322.473,-73.250,-176.537,8.056,148.560
C07055=1179.014,322.720,-73.281,-176.535,8.060,148.560
C07056=1179.010,322.968,-73.313,-176.532,8.063,148.560
C07057=1179.006,323.217,-73.344,-176.530,8.066,148.560
C07058=1179.002,323.464,-73.375,-176.527,8.069,148.560
C07059=1178.998,323.713,-73.408,-176.525,8.072,148.560
C07060=1178.993,323.960,-73.439,-176.522,8.075,148.560
C07061=1178.990,324.208,-73.471,-176.520,8.079,148.561
C07062=1178.986,324.457,-73.502,-176.517,8.082,148.561
C07063=1178.981,324.704,-73.534,-176.515,8.085,148.561
C07064=1178.977,324.953,-73.566,-176.513,8.088,148.561
C07065=1178.973,325.201,-73.598,-176.510,8.091,148.561
C07066=1178.969,325.448,-73.630,-176.508,8.095,148.561
C07067=1178.964,325.696,-73.662,-176.505,8.098,148.561
C07068=1178.961,325.944,-73.694,-176.503,8.101,148.561
C07069=1178.956,326.192,-73.725,-176.500,8.104,148.561
C07070=1178.953,326.440,-73.757,-176.498,8.107,148.562
C07071=1178.948,326.688,-73.790,-176.495,8.110,148.562
C07072=1178.944,326.936,-73.820,-176.493,8.114,148.562
C07073=1178.940,327.184,-73.852,-176.491,8.117,148.562
C07074=1178.936,327.432,-73.885,-176.488,8.120,148.562
C07075=1178.931,327.680,-73.916,-176.486,8.123,148.562
C07076=1178.928,327.927,-73.949,-176.483,8.126,148.562
C07077=1178.923,328.176,-73.981,-176.481,8.129,148.562
C07078=1178.919,328.423,-74.013,-176.478,8.133,148.563
C07079=1178.915,328.671,-74.045,-176.476,8.136,148.563
C07080=1178.911,328.919,-74.077,-176.473,8.139,148.563
C07081=1178.907,329.167,-74.108,-176.471,8.142,148.563
C07082=1178.902,329.415,-74.141,-176.468,8.145,148.563
C07083=1178.898,329.663,-74.173,-176.466,8.149,148.563
C07084=1178.894,329.911,-74.205,-176.463,8.152,148.563
C07085=1178.890,330.159,-74.237,-176.461,8.155,148.563
C07086=1178.885,330.407,-74.269,-176.458,8.158,148.563
C07087=1178.882,330.654,-74.302,-176.456,8.161,148.564
C07088=1178.878,330.902,-74.333,-176.454,8.165,148.564
C07089=1178.873,331.150,-74.366,-176.451,8.168,148.564
C07090=1178.869,331.398,-74.397,-176.449,8.171,148.564
C07091=1178.865,331.646,-74.430,-176.447,8.174,148.564
C07092=1178.861,331.893,-74.462,-176.444,8.177,148.564
C07093=1178.857,332.142,-74.494,-176.442,8.181,148.564
C07094=1178.853,332.390,-74.526,-176.439,8.184,148.565
C07095=1178.848,332.638,-74.559,-176.437,8.187,148.565
C07096=1178.845,332.885,-74.591,-176.434,8.190,148.565
C07097=1178.840,333.133,-74.623,-176.432,8.193,148.565
C07098=1178.836,333.381,-74.656,-176.429,8.196,148.565
C07099=1178.832,333.629,-74.688,-176.427,8.200,148.565
C07100=1178.828,333.877,-74.721,-176.425,8.203,148.565
C07101=1178.824,334.125,-74.753,-176.423,8.206,148.566
C07102=1178.819,334.372,-74.785,-176.420,8.209,148.566
C07103=1178.816,334.620,-74.817,-176.418,8.213,148.566
C07104=1178.811,334.869,-74.850,-176.415,8.216,148.566
C07105=1178.807,335.116,-74.883,-176.413,8.219,148.566
C07106=1178.803,335.364,-74.915,-176.410,8.222,148.566
C07107=1178.799,335.612,-74.948,-176.408,8.226,148.567
C07108=1178.795,335.859,-74.979,-176.406,8.229,148.567
C07109=1178.791,336.107,-75.013,-176.403,8.232,148.567
C07110=1178.786,336.355,-75.045,-176.401,8.235,148.567
C07111=1178.783,336.603,-75.078,-176.399,8.239,148.567
C07112=1178.778,336.851,-75.110,-176.396,8.242,148.567
C07113=1178.774,337.099,-75.143,-176.394,8.245,148.568
C07114=1178.771,337.347,-75.175,-176.391,8.248,148.568
C07115=1178.766,337.594,-75.208,-176.388,8.252,148.568
C07116=1178.761,337.842,-75.240,-176.386,8.256,148.568
C07117=1178.758,338.090,-75.273,-176.384,8.259,148.568
C07118=1178.753,338.338,-75.305,-176.381,8.262,148.568
C07119=1178.749,338.586,-75.338,-176.379,8.265,148.568
C07120=1178.745,338.834,-75.372,-176.377,8.269,148.569
C07121=1178.741,339.082,-75.403,-176.374,8.272,148.569
C07122=1178.737,339.329,-75.437,-176.372,8.275,148.569
C07123=1178.733,339.578,-75.469,-176.370,8.278,148.569
C07124=1178.728,339.856,-75.506,-176.367,8.281,148.569
C07125=1178.724,340.136,-75.543,-176.364,8.286,148.570
C07126=1178.719,340.414,-75.580,-176.362,8.290,148.570
C07127=1178.714,340.693,-75.617,-176.359,8.293,148.570
C07128=1178.710,340.941,-75.650,-176.357,8.296,148.570
C07129=1178.706,341.189,-75.682,-176.355,8.300,148.571
C07130=1178.702,341.437,-75.715,-176.352,8.303,148.571
C07131=1178.698,341.685,-75.748,-176.350,8.306,148.571
C07132=1178.694,341.932,-75.781,-176.347,8.309,148.571
C07133=1178.689,342.181,-75.814,-176.345,8.313,148.571
C07134=1178.685,342.428,-75.847,-176.342,8.317,148.571
C07135=1178.682,342.676,-75.879,-176.340,8.320,148.572
C07136=1178.678,342.924,-75.913,-176.338,8.323,148.572
C07137=1178.674,343.171,-75.946,-176.336,8.327,148.572
C07138=1178.669,343.420,-75.978,-176.333,8.330,148.572
C07139=1178.665,343.667,-76.011,-176.331,8.333,148.573
C07140=1178.661,343.915,-76.045,-176.329,8.337,148.573
C07141=1178.657,344.163,-76.078,-176.326,8.340,148.573
C07142=1178.653,344.411,-76.111,-176.324,8.343,148.573
C07143=1178.649,344.658,-76.144,-176.321,8.346,148.573
C07144=1178.644,344.906,-76.177,-176.319,8.350,148.573
C07145=1178.640,345.154,-76.210,-176.317,8.353,148.574
C07146=1178.636,345.401,-76.243,-176.315,8.356,148.574
C07147=1178.632,345.649,-76.277,-176.312,8.359,148.574
C07148=1178.629,345.897,-76.309,-176.310,8.363,148.574
C07149=1178.624,346.144,-76.342,-176.307,8.367,148.575
C07150=1178.620,346.392,-76.375,-176.305,8.370,148.575
C07151=1178.616,346.640,-76.409,-176.303,8.374,148.575
C07152=1178.612,346.887,-76.442,-176.301,8.377,148.575
C07153=1178.608,347.135,-76.475,-176.298,8.380,148.575
C07154=1178.604,347.383,-76.508,-176.296,8.384,148.576
C07155=1178.599,347.631,-76.542,-176.294,8.387,148.576
C07156=1178.595,347.879,-76.575,-176.292,8.390,148.576
C07157=1178.591,348.127,-76.609,-176.290,8.394,148.576
C07158=1178.587,348.375,-76.642,-176.287,8.397,148.577
C07159=1178.583,348.623,-76.675,-176.285,8.400,148.577
C07160=1178.579,348.870,-76.708,-176.283,8.404,148.577
C07161=1178.575,349.117,-76.742,-176.280,8.408,148.577
C07162=1178.571,349.365,-76.775,-176.278,8.411,148.578
C07163=1178.567,349.613,-76.808,-176.275,8.414,148.578
C07164=1178.563,349.861,-76.841,-176.273,8.418,148.578
C07165=1178.559,350.109,-76.875,-176.271,8.421,148.578
C07166=1178.555,350.356,-76.909,-176.269,8.425,148.579
C07167=1178.551,350.604,-76.942,-176.267,8.428,148.579
C07168=1178.546,350.852,-76.976,-176.265,8.431,148.579
C07169=1178.542,351.100,-77.009,-176.262,8.435,148.579
C07170=1178.538,351.347,-77.043,-176.260,8.438,148.580
C07171=1178.534,351.595,-77.076,-176.257,8.442,148.580
C07172=1178.531,351.843,-77.109,-176.255,8.446,148.580
C07173=1178.526,352.091,-77.143,-176.253,8.449,148.580
C07174=1178.522,352.338,-77.177,-176.251,8.452,148.581
C07175=1178.518,352.586,-77.210,-176.249,8.456,148.581
C07176=1178.514,352.834,-77.243,-176.246,8.459,148.581
C07177=1178.510,353.081,-77.277,-176.244,8.462,148.582
C07178=1178.506,353.329,-77.311,-176.242,8.466,148.582
C07179=1178.502,353.577,-77.345,-176.240,8.469,148.582
C07180=1178.497,353.824,-77.378,-176.237,8.473,148.582
C07181=1178.493,354.072,-77.411,-176.235,8.477,148.582
C07182=1178.490,354.320,-77.446,-176.233,8.480,148.583
C07183=1178.485,354.568,-77.479,-176.231,8.483,148.583
C07184=1178.481,354.815,-77.513,-176.228,8.487,148.583
C07185=1178.477,355.063,-77.546,-176.227,8.490,148.584
C07186=1178.473,355.310,-77.580,-176.224,8.494,148.584
C07187=1178.469,355.559,-77.614,-176.222,8.497,148.584
C07188=1178.465,355.806,-77.648,-176.220,8.501,148.585
C07189=1178.461,356.053,-77.681,-176.217,8.505,148.585
C07190=1178.457,356.300,-77.715,-176.215,8.508,148.585
C07191=1178.453,356.549,-77.749,-176.213,8.512,148.586
C07192=1178.449,356.796,-77.783,-176.211,8.515,148.586
C07193=1178.445,357.044,-77.816,-176.209,8.518,148.586
C07194=1178.441,357.292,-77.851,-176.207,8.522,148.586
C07195=1178.437,357.539,-77.885,-176.205,8.525,148.587
C07196=1178.433,357.787,-77.918,-176.202,8.529,148.587
C07197=1178.429,358.034,-77.953,-176.200,8.533,148.587
C07198=1178.425,358.282,-77.987,-176.198,8.536,148.588
C07199=1178.420,358.530,-78.021,-176.196,8.540,148.588
C07200=1178.417,358.777,-78.055,-176.194,8.543,148.588
C07201=1178.413,359.025,-78.089,-176.192,8.547,148.589
C07202=1178.409,359.273,-78.123,-176.190,8.550,148.589
C07203=1178.405,359.520,-78.157,-176.187,8.553,148.589
C07204=1178.401,359.768,-78.191,-176.185,8.558,148.590
C07205=1178.397,360.016,-78.225,-176.183,8.562,148.590
C07206=1178.393,360.263,-78.258,-176.181,8.565,148.590
C07207=1178.389,360.511,-78.293,-176.179,8.568,148.591
C07208=1178.385,360.759,-78.327,-176.177,8.572,148.591
C07209=1178.380,361.007,-78.361,-176.175,8.575,148.591
C07210=1178.377,361.254,-78.395,-176.173,8.579,148.592
C07211=1178.372,361.502,-78.430,-176.171,8.582,148.592
C07212=1178.368,361.749,-78.463,-176.169,8.586,148.592
C07213=1178.364,361.997,-78.498,-176.167,8.589,148.593
C07214=1178.361,362.244,-78.532,-176.165,8.593,148.593
C07215=1178.356,362.493,-78.566,-176.163,8.596,148.593
C07216=1178.353,362.740,-78.600,-176.161,8.600,148.594
C07217=1178.348,362.987,-78.635,-176.158,8.604,148.594
C07218=1178.345,363.235,-78.669,-176.157,8.608,148.595
C07219=1178.340,363.483,-78.703,-176.154,8.611,148.595
C07220=1178.337,363.730,-78.738,-176.153,8.615,148.595
C07221=1178.332,363.978,-78.772,-176.151,8.618,148.596
C07222=1178.329,364.225,-78.806,-176.149,8.622,148.596
C07223=1178.325,364.473,-78.841,-176.147,8.626,148.597
C07224=1178.321,364.720,-78.875,-176.145,8.629,148.597
C07225=1178.317,364.968,-78.909,-176.143,8.633,148.597
C07226=1178.312,365.216,-78.944,-176.141,8.636,148.598
C07227=1178.309,365.464,-78.978,-176.139,8.640,148.598
C07228=1178.304,365.745,-79.018,-176.137,8.643,148.599
C07229=1178.300,366.027,-79.056,-176.135,8.648,148.599
C07230=1178.295,366.309,-79.095,-176.133,8.651,148.599
C07231=1178.290,366.590,-79.135,-176.131,8.656,148.600
C07232=1178.287,366.838,-79.169,-176.129,8.660,148.600
C07233=1178.282,367.086,-79.203,-176.128,8.663,148.601
C07234=1178.278,367.334,-79.238,-176.126,8.667,148.601
C07235=1178.275,367.580,-79.273,-176.124,8.671,148.602
C07236=1178.271,367.828,-79.308,-176.123,8.673,148.602
C07237=1178.266,368.076,-79.342,-176.121,8.677,148.603
C07238=1178.262,368.323,-79.376,-176.119,8.681,148.603
C07239=1178.258,368.571,-79.411,-176.117,8.684,148.604
C07240=1178.254,368.818,-79.445,-176.115,8.688,148.604
C07241=1178.251,369.066,-79.480,-176.114,8.692,148.604
C07242=1178.246,369.313,-79.515,-176.112,8.695,148.605
C07243=1178.242,369.561,-79.549,-176.110,8.699,148.605
C07244=1178.238,369.809,-79.584,-176.109,8.703,148.606
C07245=1178.234,370.056,-79.618,-176.107,8.705,148.606
C07246=1178.230,370.303,-79.653,-176.106,8.709,148.607
C07247=1178.226,370.551,-79.688,-176.104,8.713,148.607
C07248=1178.222,370.799,-79.723,-176.102,8.717,148.608
C07249=1178.218,371.047,-79.757,-176.101,8.721,148.608
C07250=1178.215,371.294,-79.792,-176.100,8.723,148.609
C07251=1178.210,371.541,-79.827,-176.098,8.727,148.609
C07252=1178.206,371.790,-79.862,-176.096,8.731,148.610
C07253=1178.202,372.036,-79.897,-176.095,8.734,148.610
C07254=1178.199,372.284,-79.931,-176.094,8.738,148.611
C07255=1178.194,372.532,-79.966,-176.092,8.741,148.611
C07256=1178.190,372.779,-80.001,-176.090,8.745,148.612
C07257=1178.186,373.027,-80.036,-176.089,8.749,148.612
C07258=1178.182,373.275,-80.070,-176.088,8.752,148.613
C07259=1178.179,373.522,-80.105,-176.086,8.755,148.613
C07260=1178.174,373.769,-80.140,-176.085,8.759,148.614
C07261=1178.171,374.017,-80.175,-176.083,8.762,148.614
C07262=1178.166,374.264,-80.210,-176.082,8.766,148.615
C07263=1178.163,374.512,-80.245,-176.081,8.770,148.616
C07264=1178.159,374.760,-80.280,-176.079,8.773,148.616
C07265=1178.154,375.007,-80.315,-176.078,8.777,148.617
C07266=1178.151,375.254,-80.350,-176.076,8.780,148.617
C07267=1178.147,375.502,-80.384,-176.075,8.783,148.618
C07268=1178.143,375.749,-80.420,-176.074,8.787,148.618
C07269=1178.139,375.997,-80.455,-176.073,8.790,148.619
C07270=1178.135,376.244,-80.490,-176.071,8.794,148.619
C07271=1178.131,376.492,-80.525,-176.070,8.797,148.620
C07272=1178.126,376.739,-80.560,-176.069,8.801,148.620
C07273=1178.122,376.987,-80.595,-176.068,8.804,148.621
C07274=1178.119,377.235,-80.630,-176.067,8.808,148.622
C07275=1178.114,377.482,-80.665,-176.066,8.811,148.622
C07276=1178.111,377.730,-80.700,-176.064,8.815,148.623
C07277=1178.107,377.977,-80.736,-176.063,8.818,148.623
C07278=1178.102,378.225,-80.770,-176.062,8.822,148.624
C07279=1178.099,378.472,-80.806,-176.061,8.825,148.625
C07280=1178.095,378.720,-80.840,-176.060,8.828,148.625
C07281=1178.091,378.967,-80.875,-176.059,8.832,148.626
C07282=1178.087,379.214,-80.911,-176.058,8.835,148.626
C07283=1178.083,379.462,-80.945,-176.057,8.839,148.627
C07284=1178.079,379.709,-80.981,-176.056,8.842,148.628
C07285=1178.076,379.957,-81.016,-176.055,8.845,148.628
C07286=1178.071,380.204,-81.051,-176.054,8.848,148.629
C07287=1178.067,380.452,-81.086,-176.053,8.852,148.629
C07288=1178.064,380.699,-81.122,-176.052,8.855,148.630
C07289=1178.058,380.947,-81.157,-176.051,8.858,148.630
C07290=1178.055,381.194,-81.192,-176.050,8.862,148.631
C07291=1178.051,381.442,-81.228,-176.049,8.865,148.632
C07292=1178.047,381.690,-81.263,-176.048,8.868,148.632
C07293=1178.043,381.937,-81.298,-176.048,8.872,148.633
C07294=1178.039,382.184,-81.333,-176.047,8.875,148.634
C07295=1178.035,382.432,-81.369,-176.046,8.878,148.634
C07296=1178.031,382.679,-81.404,-176.045,8.882,148.635
C07297=1178.027,382.927,-81.439,-176.044,8.885,148.635
C07298=1178.024,383.174,-81.475,-176.043,8.888,148.636
C07299=1178.019,383.421,-81.510,-176.043,8.891,148.637
C07300=1178.015,383.669,-81.545,-176.042,8.894,148.637
C07301=1178.012,383.917,-81.580,-176.041,8.898,148.638
C07302=1178.008,384.164,-81.616,-176.041,8.901,148.639
C07303=1178.004,384.411,-81.651,-176.040,8.904,148.639
C07304=1178.000,384.658,-81.686,-176.039,8.907,148.640
C07305=1177.995,384.907,-81.722,-176.038,8.911,148.641
C07306=1177.992,385.154,-81.757,-176.038,8.914,148.641
C07307=1177.987,385.401,-81.793,-176.037,8.917,148.642
C07308=1177.984,385.649,-81.828,-176.036,8.920,148.643
C07309=1177.980,385.896,-81.864,-176.036,8.922,148.643
C07310=1177.976,386.143,-81.899,-176.036,8.926,148.644
C07311=1177.972,386.391,-81.934,-176.035,8.929,148.644
C07312=1177.968,386.639,-81.969,-176.034,8.932,148.645
C07313=1177.964,386.886,-82.005,-176.034,8.935,148.646
C07314=1177.960,387.133,-82.041,-176.033,8.938,148.646
C07315=1177.956,387.381,-82.076,-176.033,8.941,148.647
C07316=1177.952,387.628,-82.112,-176.032,8.944,148.648
C07317=1177.949,387.876,-82.147,-176.032,8.948,148.648
C07318=1177.945,388.123,-82.183,-176.032,8.950,148.649
C07319=1177.941,388.370,-82.218,-176.031,8.953,148.650
C07320=1177.936,388.618,-82.254,-176.030,8.956,148.650
C07321=1177.933,388.865,-82.290,-176.030,8.959,148.651
C07322=1177.929,389.113,-82.325,-176.030,8.962,148.652
C07323=1177.924,389.360,-82.360,-176.029,8.965,148.652
